LIN {X 0,Y 575.439,Z 360.454,A -85,B 0,C 180,E1 -10255.385,E2 -10255.385} C_VEL
LIN {X 0,Y 575.391,Z 376.581,A -85,B 0,C 180,E1 -10255.636,E2 -10255.636} C_VEL
LIN {X 0,Y 573.804,Z 481.536,A -85,B 0,C 180,E1 -10257.179,E2 -10257.179} C_VEL
LIN {X 0,Y 573.47,Z 496.036,A -85,B 0,C 180,E1 -10257.528,E2 -10257.528} C_VEL
LIN {X 0,Y 572.934,Z 510.451,A -85,B 0,C 180,E1 -10258.03,E2 -10258.03} C_VEL
LIN {X 0,Y 572.466,Z 522.841,A -85,B 0,C 180,E1 -10258.598,E2 -10258.598} C_VEL
LIN {X 0,Y 571.889,Z 535.06,A -85,B 0,C 180,E1 -10259.298,E2 -10259.298} C_VEL
LIN {X 0,Y 571.402,Z 547.39,A -85,B 0,C 180,E1 -10260.176,E2 -10260.176} C_VEL
LIN {X 0,Y 570.935,Z 557.583,A -85,B 0,C 180,E1 -10261.054,E2 -10261.054} C_VEL
LIN {X 0,Y 570.32,Z 567.822,A -85,B 0,C 180,E1 -10262.112,E2 -10262.112} C_VEL
LIN {X 0,Y 569.977,Z 576.267,A -85,B 0,C 180,E1 -10263.17,E2 -10263.17} C_VEL
LIN {X 0,Y 569.621,Z 583.313,A -85,B 0,C 180,E1 -10264.231,E2 -10264.231} C_VEL
LIN {X 0,Y 569.503,Z 588.963,A -85,B 0,C 180,E1 -10265.257,E2 -10265.257} C_VEL
LIN {X 0,Y 569.323,Z 593.962,A -85,B 0,C 180,E1 -10266.357,E2 -10266.357} C_VEL
LIN {X 0,Y 569.1,Z 598.933,A -85,B 0,C 180,E1 -10267.781,E2 -10267.781} C_VEL
LIN {X 0,Y 569.035,Z 602.372,A -85,B 0,C 180,E1 -10269.208,E2 -10269.208} C_VEL
LIN {X 0,Y 569.056,Z 603.678,A -85,B 0,C 180,E1 -10270.028,E2 -10270.028} C_VEL
LIN {X 0,Y 568.925,Z 604.796,A -85,B 0,C 180,E1 -10271.361,E2 -10271.361} C_VEL
LIN {X 0,Y 568.971,Z 604.604,A -85,B 0,C 180,E1 -10272.803,E2 -10272.803} C_VEL
LIN {X 0,Y 569.033,Z 603.97,A -85,B 0,C 180,E1 -10273.526,E2 -10273.526} C_VEL
LIN {X 0,Y 568.978,Z 601.595,A -85,B 0,C 180,E1 -10274.982,E2 -10274.982} C_VEL
LIN {X 0,Y 569.112,Z 597.684,A -85,B 0,C 180,E1 -10276.444,E2 -10276.444} C_VEL
LIN {X 0,Y 569.206,Z 593.593,A -85,B 0,C 180,E1 -10277.547,E2 -10277.547} C_VEL
LIN {X 0,Y 569.387,Z 588.256,A -85,B 0,C 180,E1 -10278.693,E2 -10278.693} C_VEL
LIN {X 0,Y 569.633,Z 580.967,A -85,B 0,C 180,E1 -10279.952,E2 -10279.952} C_VEL
LIN {X 0,Y 569.942,Z 573.158,A -85,B 0,C 180,E1 -10281.049,E2 -10281.049} C_VEL
LIN {X 0,Y 570.356,Z 563.337,A -85,B 0,C 180,E1 -10282.187,E2 -10282.187} C_VEL
LIN {X 0,Y 570.787,Z 552.451,A -85,B 0,C 180,E1 -10283.218,E2 -10283.218} C_VEL
LIN {X 0,Y 571.326,Z 540.367,A -85,B 0,C 180,E1 -10284.153,E2 -10284.153} C_VEL
LIN {X 0,Y 571.808,Z 527.265,A -85,B 0,C 180,E1 -10284.976,E2 -10284.976} C_VEL
LIN {X 0,Y 572.223,Z 514.526,A -85,B 0,C 180,E1 -10285.611,E2 -10285.611} C_VEL
LIN {X 0,Y 572.651,Z 501.122,A -85,B 0,C 180,E1 -10286.125,E2 -10286.125} C_VEL
LIN {X 0,Y 573.109,Z 487.002,A -85,B 0,C 180,E1 -10286.518,E2 -10286.518} C_VEL
LIN {X 0,Y 573.287,Z 471.7,A -85,B 0,C 180,E1 -10286.795,E2 -10286.795} C_VEL
LIN {X 0,Y 574.437,Z 360.487,A -85,B 0,C 180,E1 -10288.346,E2 -10288.346} C_VEL
LIN {X 0,Y 571.59,Z 342.196,A -85,B 0,C 180,E1 -10288.699,E2 -10288.699} C_VEL
LIN {X 0,Y 572.257,Z 318.728,A -85,B 0,C 180,E1 -10291.757,E2 -10291.757} C_VEL
LIN {X 0,Y 572.767,Z 299.778,A -85,B 0,C 180,E1 -10294.232,E2 -10294.232} C_VEL
LIN {X 0,Y 571.08,Z 289.612,A -85,B 0,C 180,E1 -10295.634,E2 -10295.634} C_VEL
LIN {X 0,Y 570.357,Z 286,A -85,B 0,C 180,E1 -10296.147,E2 -10296.147} C_VEL
LIN {X 0,Y 570.263,Z 286.005,A -85,B 0,C 180,E1 -10299.3,E2 -10299.3} C_VEL
LIN {X 0,Y 570.28,Z 286.004,A -85,B 0,C 180,E1 -10301.548,E2 -10301.548} C_VEL
LIN {X 0,Y 570.317,Z 286.001,A -85,B 0,C 180,E1 -10304.573,E2 -10304.573} C_VEL
LIN {X 0,Y 570.263,Z 286.007,A -85,B 0,C 180,E1 -10307.501,E2 -10307.501} C_VEL
LIN {X 0,Y 570.283,Z 286.006,A -85,B 0,C 180,E1 -10310.305,E2 -10310.305} C_VEL
LIN {X 0,Y 570.273,Z 286.007,A -85,B 0,C 180,E1 -10312.996,E2 -10312.996} C_VEL
LIN {X 0,Y 570.287,Z 286.006,A -85,B 0,C 180,E1 -10315.597,E2 -10315.597} C_VEL
LIN {X 0,Y 570.315,Z 286.001,A -85,B 0,C 180,E1 -10318.121,E2 -10318.121} C_VEL
LIN {X 0,Y 570.294,Z 286.005,A -85,B 0,C 180,E1 -10321.378,E2 -10321.378} C_VEL
LIN {X 0,Y 570.293,Z 286.004,A -85,B 0,C 180,E1 -10322.089,E2 -10322.089} C_VEL
LIN {X 0,Y 569.657,Z 286.086,A -85,B 0,C 180,E1 -10322.678,E2 -10322.678} C_VEL
LIN {X 0,Y 566.811,Z 286.439,A -85,B 0,C 180,E1 -10323.635,E2 -10323.635} C_VEL
LIN {X 0,Y 564.388,Z 286.742,A -85,B 0,C 180,E1 -10324.404,E2 -10324.404} C_VEL
LIN {X 0,Y 563.349,Z 286.869,A -85,B 0,C 180,E1 -10324.999,E2 -10324.999} C_VEL
LIN {X 0,Y 563.267,Z 286.879,A -85,B 0,C 180,E1 -10325.2,E2 -10325.2} C_VEL
LIN {X 0,Y 563.302,Z 286.876,A -85,B 0,C 180,E1 -10328.095,E2 -10328.095} C_VEL
LIN {X 0,Y 563.305,Z 286.874,A -85,B 0,C 180,E1 -10331.136,E2 -10331.136} C_VEL
LIN {X 0,Y 563.311,Z 286.878,A -85,B 0,C 180,E1 -10334.122,E2 -10334.122} C_VEL
LIN {X 0,Y 563.359,Z 286.869,A -85,B 0,C 180,E1 -10336.334,E2 -10336.334} C_VEL
LIN {X 0,Y 563.372,Z 286.864,A -85,B 0,C 180,E1 -10339.25,E2 -10339.25} C_VEL
LIN {X 0,Y 563.397,Z 286.866,A -85,B 0,C 180,E1 -10342.497,E2 -10342.497} C_VEL
LIN {X 0,Y 563.431,Z 286.922,A -85,B 0,C 180,E1 -10342.857,E2 -10342.857} C_VEL
LIN {X 0,Y 564.572,Z 294.675,A -85,B 0,C 180,E1 -10344.302,E2 -10344.302} C_VEL
LIN {X 0,Y 564.436,Z 300.116,A -85,B 0,C 180,E1 -10345.271,E2 -10345.271} C_VEL
LIN {X 0,Y 567.828,Z 316.778,A -85,B 0,C 180,E1 -10345.577,E2 -10345.577} C_VEL
LIN {X 0,Y 566.808,Z 435.74,A -85,B 0,C 180,E1 -10347.099,E2 -10347.099} C_VEL
LIN {X 0,Y 566.508,Z 450.139,A -85,B 0,C 180,E1 -10347.429,E2 -10347.429} C_VEL
LIN {X 0,Y 566.207,Z 463.339,A -85,B 0,C 180,E1 -10347.871,E2 -10347.871} C_VEL
LIN {X 0,Y 565.821,Z 475.423,A -85,B 0,C 180,E1 -10348.402,E2 -10348.402} C_VEL
LIN {X 0,Y 565.416,Z 488.106,A -85,B 0,C 180,E1 -10349.111,E2 -10349.111} C_VEL
LIN {X 0,Y 564.727,Z 499.728,A -85,B 0,C 180,E1 -10349.909,E2 -10349.909} C_VEL
LIN {X 0,Y 564.286,Z 511.265,A -85,B 0,C 180,E1 -10350.887,E2 -10350.887} C_VEL
LIN {X 0,Y 563.681,Z 521.642,A -85,B 0,C 180,E1 -10351.957,E2 -10351.957} C_VEL
LIN {X 0,Y 563.288,Z 530.194,A -85,B 0,C 180,E1 -10353.028,E2 -10353.028} C_VEL
LIN {X 0,Y 562.818,Z 538.433,A -85,B 0,C 180,E1 -10354.281,E2 -10354.281} C_VEL
LIN {X 0,Y 562.684,Z 544.812,A -85,B 0,C 180,E1 -10355.488,E2 -10355.488} C_VEL
LIN {X 0,Y 562.439,Z 550.296,A -85,B 0,C 180,E1 -10356.793,E2 -10356.793} C_VEL
LIN {X 0,Y 562.242,Z 553.805,A -85,B 0,C 180,E1 -10357.875,E2 -10357.875} C_VEL
LIN {X 0,Y 562.144,Z 557.231,A -85,B 0,C 180,E1 -10359.32,E2 -10359.32} C_VEL
LIN {X 0,Y 562.095,Z 559.271,A -85,B 0,C 180,E1 -10360.771,E2 -10360.771} C_VEL
LIN {X 0,Y 562.043,Z 559.951,A -85,B 0,C 180,E1 -10362.229,E2 -10362.229} C_VEL
LIN {X 0,Y 562.154,Z 559.253,A -85,B 0,C 180,E1 -10363.692,E2 -10363.692} C_VEL
LIN {X 0,Y 562.211,Z 557.174,A -85,B 0,C 180,E1 -10365.165,E2 -10365.165} C_VEL
LIN {X 0,Y 562.424,Z 553.635,A -85,B 0,C 180,E1 -10366.643,E2 -10366.643} C_VEL
LIN {X 0,Y 562.685,Z 548.511,A -85,B 0,C 180,E1 -10368.13,E2 -10368.13} C_VEL
LIN {X 0,Y 563.038,Z 542.646,A -85,B 0,C 180,E1 -10369.418,E2 -10369.418} C_VEL
LIN {X 0,Y 563.498,Z 535.031,A -85,B 0,C 180,E1 -10370.746,E2 -10370.746} C_VEL
LIN {X 0,Y 564.017,Z 527.054,A -85,B 0,C 180,E1 -10371.872,E2 -10371.872} C_VEL
LIN {X 0,Y 564.601,Z 517.329,A -85,B 0,C 180,E1 -10373.001,E2 -10373.001} C_VEL
LIN {X 0,Y 565.263,Z 506.553,A -85,B 0,C 180,E1 -10374.028,E2 -10374.028} C_VEL
LIN {X 0,Y 565.934,Z 494.604,A -85,B 0,C 180,E1 -10374.958,E2 -10374.958} C_VEL
LIN {X 0,Y 566.519,Z 482.243,A -85,B 0,C 180,E1 -10375.737,E2 -10375.737} C_VEL
LIN {X 0,Y 567.105,Z 468.979,A -85,B 0,C 180,E1 -10376.398,E2 -10376.398} C_VEL
LIN {X 0,Y 567.526,Z 456.619,A -85,B 0,C 180,E1 -10376.871,E2 -10376.871} C_VEL
LIN {X 0,Y 567.835,Z 442.693,A -85,B 0,C 180,E1 -10377.263,E2 -10377.263} C_VEL
LIN {X 0,Y 567.93,Z 427.921,A -85,B 0,C 180,E1 -10377.524,E2 -10377.524} C_VEL
LIN {X 0,Y 569.043,Z 317.141,A -85,B 0,C 180,E1 -10378.943,E2 -10378.943} C_VEL
LIN {X 0,Y 565.232,Z 300.482,A -85,B 0,C 180,E1 -10379.325,E2 -10379.325} C_VEL
LIN {X 0,Y 565.026,Z 296.096,A -85,B 0,C 180,E1 -10380.146,E2 -10380.146} C_VEL
LIN {X 0,Y 563.228,Z 286.887,A -85,B 0,C 180,E1 -10381.992,E2 -10381.992} C_VEL
LIN {X 0,Y 563.243,Z 286.882,A -85,B 0,C 180,E1 -10384.891,E2 -10384.891} C_VEL
LIN {X 0,Y 563.207,Z 286.886,A -85,B 0,C 180,E1 -10387.543,E2 -10387.543} C_VEL
LIN {X 0,Y 563.226,Z 286.882,A -85,B 0,C 180,E1 -10390.658,E2 -10390.658} C_VEL
LIN {X 0,Y 563.238,Z 286.882,A -85,B 0,C 180,E1 -10393.152,E2 -10393.152} C_VEL
LIN {X 0,Y 563.232,Z 286.879,A -85,B 0,C 180,E1 -10395.859,E2 -10395.859} C_VEL
LIN {X 0,Y 563.227,Z 286.882,A -85,B 0,C 180,E1 -10398.767,E2 -10398.767} C_VEL
LIN {X 0,Y 563.249,Z 286.883,A -85,B 0,C 180,E1 -10401.574,E2 -10401.574} C_VEL
LIN {X 0,Y 563.273,Z 286.863,A -85,B 0,C 180,E1 -10404.235,E2 -10404.235} C_VEL
LIN {X 0,Y 563.205,Z 286.883,A -85,B 0,C 180,E1 -10406.824,E2 -10406.824} C_VEL
LIN {X 0,Y 563.26,Z 286.877,A -85,B 0,C 180,E1 -10409.346,E2 -10409.346} C_VEL
LIN {X 0,Y 563.269,Z 286.875,A -85,B 0,C 180,E1 -10411.99,E2 -10411.99} C_VEL
LIN {X 0,Y 563.24,Z 286.883,A -85,B 0,C 180,E1 -10415.201,E2 -10415.201} C_VEL
LIN {X 0,Y 563.275,Z 286.876,A -85,B 0,C 180,E1 -10418.096,E2 -10418.096} C_VEL
LIN {X 0,Y 563.274,Z 286.874,A -85,B 0,C 180,E1 -10421.136,E2 -10421.136} C_VEL
LIN {X 0,Y 563.269,Z 286.875,A -85,B 0,C 180,E1 -10424.123,E2 -10424.123} C_VEL
LIN {X 0,Y 563.341,Z 286.86,A -85,B 0,C 180,E1 -10426.335,E2 -10426.335} C_VEL
LIN {X 0,Y 563.343,Z 286.873,A -85,B 0,C 180,E1 -10429.251,E2 -10429.251} C_VEL
LIN {X 0,Y 563.367,Z 286.86,A -85,B 0,C 180,E1 -10432.139,E2 -10432.139} C_VEL
LIN {X 0,Y 563.439,Z 286.86,A -85,B 0,C 180,E1 -10435.008,E2 -10435.008} C_VEL
LIN {X 0,Y 563.447,Z 286.854,A -85,B 0,C 180,E1 -10438.575,E2 -10438.575} C_VEL
LIN {X 0,Y 563.573,Z 286.836,A -85,B 0,C 180,E1 -10440,E2 -10440} C_VEL
LIN {X 0,Y 563.303,Z 286.862,A -85,B 0,C 180,E1 -10442.138,E2 -10442.138} C_VEL
LIN {X 0,Y 563.455,Z 286.86,A -85,B 0,C 180,E1 -10444.992,E2 -10444.992} C_VEL
LIN {X 0,Y 563.368,Z 286.855,A -85,B 0,C 180,E1 -10447.861,E2 -10447.861} C_VEL
LIN {X 0,Y 563.392,Z 286.864,A -85,B 0,C 180,E1 -10450.848,E2 -10450.848} C_VEL
LIN {X 0,Y 563.349,Z 286.862,A -85,B 0,C 180,E1 -10454.123,E2 -10454.123} C_VEL
LIN {X 0,Y 563.319,Z 286.868,A -85,B 0,C 180,E1 -10456.786,E2 -10456.786} C_VEL
LIN {X 0,Y 563.26,Z 286.875,A -85,B 0,C 180,E1 -10459.619,E2 -10459.619} C_VEL
LIN {X 0,Y 563.275,Z 286.869,A -85,B 0,C 180,E1 -10461.904,E2 -10461.904} C_VEL
LIN {X 0,Y 563.24,Z 286.883,A -85,B 0,C 180,E1 -10464.8,E2 -10464.8} C_VEL
LIN {X 0,Y 563.269,Z 286.876,A -85,B 0,C 180,E1 -10468.01,E2 -10468.01} C_VEL
LIN {X 0,Y 563.261,Z 286.879,A -85,B 0,C 180,E1 -10470.907,E2 -10470.907} C_VEL
LIN {X 0,Y 563.237,Z 286.877,A -85,B 0,C 180,E1 -10473.574,E2 -10473.574} C_VEL
LIN {X 0,Y 563.309,Z 286.856,A -85,B 0,C 180,E1 -10476.08,E2 -10476.08} C_VEL
LIN {X 0,Y 563.3,Z 286.879,A -85,B 0,C 180,E1 -10478.443,E2 -10478.443} C_VEL
LIN {X 0,Y 563.243,Z 286.879,A -85,B 0,C 180,E1 -10481.232,E2 -10481.232} C_VEL
LIN {X 0,Y 563.228,Z 286.883,A -85,B 0,C 180,E1 -10483.841,E2 -10483.841} C_VEL
LIN {X 0,Y 563.233,Z 286.887,A -85,B 0,C 180,E1 -10486.162,E2 -10486.162} C_VEL
LIN {X 0,Y 563.264,Z 286.877,A -85,B 0,C 180,E1 -10488.773,E2 -10488.773} C_VEL
LIN {X 0,Y 563.285,Z 286.876,A -85,B 0,C 180,E1 -10491.573,E2 -10491.573} C_VEL
LIN {X 0,Y 563.303,Z 286.877,A -85,B 0,C 180,E1 -10494.24,E2 -10494.24} C_VEL
LIN {X 0,Y 563.244,Z 286.884,A -85,B 0,C 180,E1 -10496.829,E2 -10496.829} C_VEL
LIN {X 0,Y 563.266,Z 286.884,A -85,B 0,C 180,E1 -10499.349,E2 -10499.349} C_VEL
LIN {X 0,Y 563.289,Z 286.879,A -85,B 0,C 180,E1 -10502.516,E2 -10502.516} C_VEL
LIN {X 0,Y 566.847,Z 303.208,A -85,B 0,C 180,E1 -10505.009,E2 -10505.009} C_VEL
LIN {X 0,Y 567.241,Z 307.117,A -85,B 0,C 180,E1 -10505.567,E2 -10505.567} C_VEL
LIN {X 0,Y 566.095,Z 326.832,A -85,B 0,C 180,E1 -10508.213,E2 -10508.213} C_VEL
LIN {X 0,Y 564.836,Z 350.849,A -85,B 0,C 180,E1 -10511.38,E2 -10511.38} C_VEL
LIN {X 0,Y 564.394,Z 361.151,A -85,B 0,C 180,E1 -10512.71,E2 -10512.71} C_VEL
LIN {X 0,Y 567.671,Z 382.814,A -85,B 0,C 180,E1 -10513.112,E2 -10513.112} C_VEL
LIN {X 0,Y 568.575,Z 391.391,A -85,B 0,C 180,E1 -10513.255,E2 -10513.255} C_VEL
LIN {X 0,Y 567.497,Z 499.318,A -85,B 0,C 180,E1 -10514.651,E2 -10514.651} C_VEL
LIN {X 0,Y 566.972,Z 514.115,A -85,B 0,C 180,E1 -10514.988,E2 -10514.988} C_VEL
LIN {X 0,Y 566.391,Z 527.966,A -85,B 0,C 180,E1 -10515.453,E2 -10515.453} C_VEL
LIN {X 0,Y 565.747,Z 540.9,A -85,B 0,C 180,E1 -10516.031,E2 -10516.031} C_VEL
LIN {X 0,Y 565.032,Z 553.471,A -85,B 0,C 180,E1 -10516.744,E2 -10516.744} C_VEL
LIN {X 0,Y 564.367,Z 564.958,A -85,B 0,C 180,E1 -10517.549,E2 -10517.549} C_VEL
LIN {X 0,Y 563.709,Z 576.506,A -85,B 0,C 180,E1 -10518.535,E2 -10518.535} C_VEL
LIN {X 0,Y 563.228,Z 586.869,A -85,B 0,C 180,E1 -10519.613,E2 -10519.613} C_VEL
LIN {X 0,Y 562.765,Z 595.446,A -85,B 0,C 180,E1 -10520.69,E2 -10520.69} C_VEL
LIN {X 0,Y 562.348,Z 603.685,A -85,B 0,C 180,E1 -10521.947,E2 -10521.947} C_VEL
LIN {X 0,Y 562.143,Z 612.58,A -85,B 0,C 180,E1 -10523.563,E2 -10523.563} C_VEL
LIN {X 0,Y 562.068,Z 617.376,A -85,B 0,C 180,E1 -10524.639,E2 -10524.639} C_VEL
LIN {X 0,Y 561.972,Z 621.998,A -85,B 0,C 180,E1 -10525.971,E2 -10525.971} C_VEL
LIN {X 0,Y 562.009,Z 624.928,A -85,B 0,C 180,E1 -10527.144,E2 -10527.144} C_VEL
LIN {X 0,Y 561.962,Z 627.166,A -85,B 0,C 180,E1 -10528.573,E2 -10528.573} C_VEL
LIN {X 0,Y 561.985,Z 627.985,A -85,B 0,C 180,E1 -10530.002,E2 -10530.002} C_VEL
LIN {X 0,Y 561.961,Z 627.392,A -85,B 0,C 180,E1 -10531.43,E2 -10531.43} C_VEL
LIN {X 0,Y 562.011,Z 625.363,A -85,B 0,C 180,E1 -10532.859,E2 -10532.859} C_VEL
LIN {X 0,Y 562.019,Z 621.854,A -85,B 0,C 180,E1 -10534.29,E2 -10534.29} C_VEL
LIN {X 0,Y 562.073,Z 618.238,A -85,B 0,C 180,E1 -10535.365,E2 -10535.365} C_VEL
LIN {X 0,Y 562.151,Z 613.624,A -85,B 0,C 180,E1 -10536.44,E2 -10536.44} C_VEL
LIN {X 0,Y 562.339,Z 606.953,A -85,B 0,C 180,E1 -10537.697,E2 -10537.697} C_VEL
LIN {X 0,Y 562.664,Z 598.641,A -85,B 0,C 180,E1 -10538.954,E2 -10538.954} C_VEL
LIN {X 0,Y 562.963,Z 589.911,A -85,B 0,C 180,E1 -10540.033,E2 -10540.033} C_VEL
LIN {X 0,Y 563.464,Z 580.417,A -85,B 0,C 180,E1 -10541.011,E2 -10541.011} C_VEL
LIN {X 0,Y 563.945,Z 568.675,A -85,B 0,C 180,E1 -10542.009,E2 -10542.009} C_VEL
LIN {X 0,Y 564.465,Z 557.07,A -85,B 0,C 180,E1 -10542.817,E2 -10542.817} C_VEL
LIN {X 0,Y 565.06,Z 544.353,A -85,B 0,C 180,E1 -10543.533,E2 -10543.533} C_VEL
LIN {X 0,Y 565.545,Z 531.258,A -85,B 0,C 180,E1 -10544.115,E2 -10544.115} C_VEL
LIN {X 0,Y 566.049,Z 517.241,A -85,B 0,C 180,E1 -10544.582,E2 -10544.582} C_VEL
LIN {X 0,Y 566.5,Z 499.468,A -85,B 0,C 180,E1 -10544.982,E2 -10544.982} C_VEL
LIN {X 0,Y 567.554,Z 424.5,A -85,B 0,C 180,E1 -10546.077,E2 -10546.077} C_VEL
LIN {X 0,Y 568.068,Z 389.136,A -85,B 0,C 180,E1 -10546.623,E2 -10546.623} C_VEL
LIN {X 0,Y 564.86,Z 363.019,A -85,B 0,C 180,E1 -10547.174,E2 -10547.174} C_VEL
LIN {X 0,Y 564.089,Z 357.909,A -85,B 0,C 180,E1 -10547.295,E2 -10547.295} C_VEL
LIN {X 0,Y 564.97,Z 335.865,A -85,B 0,C 180,E1 -10550.125,E2 -10550.125} C_VEL
LIN {X 0,Y 566.057,Z 312.595,A -85,B 0,C 180,E1 -10553.135,E2 -10553.135} C_VEL
LIN {X 0,Y 566.375,Z 302.386,A -85,B 0,C 180,E1 -10554.477,E2 -10554.477} C_VEL
LIN {X 0,Y 563.285,Z 286.88,A -85,B 0,C 180,E1 -10556.695,E2 -10556.695} C_VEL
LIN {X 0,Y 563.254,Z 286.883,A -85,B 0,C 180,E1 -10559.483,E2 -10559.483} C_VEL
LIN {X 0,Y 563.247,Z 286.878,A -85,B 0,C 180,E1 -10562.328,E2 -10562.328} C_VEL
LIN {X 0,Y 563.261,Z 286.879,A -85,B 0,C 180,E1 -10564.894,E2 -10564.894} C_VEL
LIN {X 0,Y 563.204,Z 286.892,A -85,B 0,C 180,E1 -10567.548,E2 -10567.548} C_VEL
LIN {X 0,Y 563.245,Z 286.88,A -85,B 0,C 180,E1 -10570.66,E2 -10570.66} C_VEL
LIN {X 0,Y 563.226,Z 286.883,A -85,B 0,C 180,E1 -10573.838,E2 -10573.838} C_VEL
LIN {X 0,Y 563.24,Z 286.88,A -85,B 0,C 180,E1 -10576.162,E2 -10576.162} C_VEL
LIN {X 0,Y 563.246,Z 286.882,A -85,B 0,C 180,E1 -10579.341,E2 -10579.341} C_VEL
LIN {X 0,Y 563.227,Z 286.886,A -85,B 0,C 180,E1 -10582.455,E2 -10582.455} C_VEL
LIN {X 0,Y 563.276,Z 286.879,A -85,B 0,C 180,E1 -10585.159,E2 -10585.159} C_VEL
LIN {X 0,Y 563.252,Z 286.879,A -85,B 0,C 180,E1 -10587.741,E2 -10587.741} C_VEL
LIN {X 0,Y 563.257,Z 286.884,A -85,B 0,C 180,E1 -10590.518,E2 -10590.518} C_VEL
LIN {X 0,Y 563.276,Z 286.881,A -85,B 0,C 180,E1 -10592.606,E2 -10592.606} C_VEL
LIN {X 0,Y 563.268,Z 286.882,A -85,B 0,C 180,E1 -10595.772,E2 -10595.772} C_VEL
LIN {X 0,Y 563.305,Z 286.883,A -85,B 0,C 180,E1 -10598.097,E2 -10598.097} C_VEL
LIN {X 0,Y 563.305,Z 286.879,A -85,B 0,C 180,E1 -10601.137,E2 -10601.137} C_VEL
LIN {X 0,Y 563.291,Z 286.879,A -85,B 0,C 180,E1 -10604.123,E2 -10604.123} C_VEL
LIN {X 0,Y 563.362,Z 286.871,A -85,B 0,C 180,E1 -10606.336,E2 -10606.336} C_VEL
LIN {X 0,Y 563.322,Z 286.946,A -85,B 0,C 180,E1 -10607.272,E2 -10607.272} C_VEL
LIN {X 0,Y 566.211,Z 300.084,A -85,B 0,C 180,E1 -10609.126,E2 -10609.126} C_VEL
LIN {X 0,Y 566.493,Z 305.5,A -85,B 0,C 180,E1 -10609.852,E2 -10609.852} C_VEL
LIN {X 0,Y 566.027,Z 325.116,A -85,B 0,C 180,E1 -10612.38,E2 -10612.38} C_VEL
LIN {X 0,Y 565.383,Z 343.211,A -85,B 0,C 180,E1 -10614.713,E2 -10614.713} C_VEL
LIN {X 0,Y 568.329,Z 358.791,A -85,B 0,C 180,E1 -10615.095,E2 -10615.095} C_VEL
LIN {X 0,Y 568.96,Z 363.16,A -85,B 0,C 180,E1 -10615.189,E2 -10615.189} C_VEL
LIN {X 0,Y 566.993,Z 482.592,A -85,B 0,C 180,E1 -10616.99,E2 -10616.99} C_VEL
LIN {X 0,Y 566.647,Z 496.712,A -85,B 0,C 180,E1 -10617.343,E2 -10617.343} C_VEL
LIN {X 0,Y 566.103,Z 510.414,A -85,B 0,C 180,E1 -10617.828,E2 -10617.828} C_VEL
LIN {X 0,Y 565.619,Z 522.816,A -85,B 0,C 180,E1 -10618.403,E2 -10618.403} C_VEL
LIN {X 0,Y 565.016,Z 535.052,A -85,B 0,C 180,E1 -10619.112,E2 -10619.112} C_VEL
LIN {X 0,Y 564.472,Z 547.43,A -85,B 0,C 180,E1 -10620,E2 -10620} C_VEL
LIN {X 0,Y 563.987,Z 557.648,A -85,B 0,C 180,E1 -10620.889,E2 -10620.889} C_VEL
LIN {X 0,Y 563.341,Z 567.899,A -85,B 0,C 180,E1 -10621.959,E2 -10621.959} C_VEL
LIN {X 0,Y 562.98,Z 576.351,A -85,B 0,C 180,E1 -10623.031,E2 -10623.031} C_VEL
LIN {X 0,Y 562.559,Z 583.414,A -85,B 0,C 180,E1 -10624.105,E2 -10624.105} C_VEL
LIN {X 0,Y 562.426,Z 590.153,A -85,B 0,C 180,E1 -10625.359,E2 -10625.359} C_VEL
LIN {X 0,Y 562.248,Z 594.798,A -85,B 0,C 180,E1 -10626.438,E2 -10626.438} C_VEL
LIN {X 0,Y 562,Z 599.608,A -85,B 0,C 180,E1 -10627.88,E2 -10627.88} C_VEL
LIN {X 0,Y 561.951,Z 602.845,A -85,B 0,C 180,E1 -10629.325,E2 -10629.325} C_VEL
LIN {X 0,Y 561.981,Z 603.908,A -85,B 0,C 180,E1 -10630.049,E2 -10630.049} C_VEL
LIN {X 0,Y 561.835,Z 604.982,A -85,B 0,C 180,E1 -10631.506,E2 -10631.506} C_VEL
LIN {X 0,Y 561.895,Z 604.625,A -85,B 0,C 180,E1 -10632.967,E2 -10632.967} C_VEL
LIN {X 0,Y 561.926,Z 603.906,A -85,B 0,C 180,E1 -10633.7,E2 -10633.7} C_VEL
LIN {X 0,Y 561.893,Z 601.356,A -85,B 0,C 180,E1 -10635.176,E2 -10635.176} C_VEL
LIN {X 0,Y 562.031,Z 598.235,A -85,B 0,C 180,E1 -10636.333,E2 -10636.333} C_VEL
LIN {X 0,Y 562.172,Z 592.965,A -85,B 0,C 180,E1 -10637.774,E2 -10637.774} C_VEL
LIN {X 0,Y 562.418,Z 586.621,A -85,B 0,C 180,E1 -10639.082,E2 -10639.082} C_VEL
LIN {X 0,Y 562.606,Z 579.844,A -85,B 0,C 180,E1 -10640.212,E2 -10640.212} C_VEL
LIN {X 0,Y 562.972,Z 571.595,A -85,B 0,C 180,E1 -10641.341,E2 -10641.341} C_VEL
LIN {X 0,Y 563.415,Z 561.525,A -85,B 0,C 180,E1 -10642.475,E2 -10642.475} C_VEL
LIN {X 0,Y 563.868,Z 550.24,A -85,B 0,C 180,E1 -10643.519,E2 -10643.519} C_VEL
LIN {X 0,Y 564.359,Z 538.998,A -85,B 0,C 180,E1 -10644.373,E2 -10644.373} C_VEL
LIN {X 0,Y 564.845,Z 526.629,A -85,B 0,C 180,E1 -10645.141,E2 -10645.141} C_VEL
LIN {X 0,Y 565.291,Z 513.254,A -85,B 0,C 180,E1 -10645.8,E2 -10645.8} C_VEL
LIN {X 0,Y 565.727,Z 499.409,A -85,B 0,C 180,E1 -10646.321,E2 -10646.321} C_VEL
LIN {X 0,Y 566.171,Z 484.533,A -85,B 0,C 180,E1 -10646.72,E2 -10646.72} C_VEL
LIN {X 0,Y 566.376,Z 467.777,A -85,B 0,C 180,E1 -10646.998,E2 -10646.998} C_VEL
LIN {X 0,Y 567.563,Z 361.331,A -85,B 0,C 180,E1 -10648.508,E2 -10648.508} C_VEL
LIN {X 0,Y 564.62,Z 342.226,A -85,B 0,C 180,E1 -10648.887,E2 -10648.887} C_VEL
LIN {X 0,Y 565.275,Z 320.222,A -85,B 0,C 180,E1 -10651.778,E2 -10651.778} C_VEL
LIN {X 0,Y 565.83,Z 301.104,A -85,B 0,C 180,E1 -10654.289,E2 -10654.289} C_VEL
LIN {X 0,Y 563.894,Z 289.819,A -85,B 0,C 180,E1 -10655.85,E2 -10655.85} C_VEL
LIN {X 0,Y 563.304,Z 286.879,A -85,B 0,C 180,E1 -10656.295,E2 -10656.295} C_VEL
LIN {X 0,Y 563.234,Z 286.882,A -85,B 0,C 180,E1 -10659.551,E2 -10659.551} C_VEL
LIN {X 0,Y 563.269,Z 286.883,A -85,B 0,C 180,E1 -10662.184,E2 -10662.184} C_VEL
LIN {X 0,Y 563.278,Z 286.877,A -85,B 0,C 180,E1 -10665.138,E2 -10665.138} C_VEL
LIN {X 0,Y 563.212,Z 286.887,A -85,B 0,C 180,E1 -10668.262,E2 -10668.262} C_VEL
LIN {X 0,Y 563.219,Z 286.885,A -85,B 0,C 180,E1 -10670.634,E2 -10670.634} C_VEL
LIN {X 0,Y 563.257,Z 286.883,A -85,B 0,C 180,E1 -10673.932,E2 -10673.932} C_VEL
LIN {X 0,Y 563.228,Z 286.885,A -85,B 0,C 180,E1 -10676.824,E2 -10676.824} C_VEL
LIN {X 0,Y 563.25,Z 286.882,A -85,B 0,C 180,E1 -10679.344,E2 -10679.344} C_VEL
LIN {X 0,Y 563.264,Z 286.879,A -85,B 0,C 180,E1 -10682.085,E2 -10682.085} C_VEL
LIN {X 0,Y 563.267,Z 286.879,A -85,B 0,C 180,E1 -10685.2,E2 -10685.2} C_VEL
LIN {X 0,Y 562.602,Z 286.963,A -85,B 0,C 180,E1 -10685.797,E2 -10685.797} C_VEL
LIN {X 0,Y 559.742,Z 287.318,A -85,B 0,C 180,E1 -10686.765,E2 -10686.765} C_VEL
LIN {X 0,Y 557.333,Z 287.618,A -85,B 0,C 180,E1 -10687.545,E2 -10687.545} C_VEL
LIN {X 0,Y 556.313,Z 287.747,A -85,B 0,C 180,E1 -10688.147,E2 -10688.147} C_VEL
LIN {X 0,Y 556.237,Z 287.754,A -85,B 0,C 180,E1 -10688.351,E2 -10688.351} C_VEL
LIN {X 0,Y 556.252,Z 287.752,A -85,B 0,C 180,E1 -10690.888,E2 -10690.888} C_VEL
LIN {X 0,Y 556.264,Z 287.753,A -85,B 0,C 180,E1 -10693.916,E2 -10693.916} C_VEL
LIN {X 0,Y 556.328,Z 287.747,A -85,B 0,C 180,E1 -10696.158,E2 -10696.158} C_VEL
LIN {X 0,Y 556.361,Z 287.737,A -85,B 0,C 180,E1 -10699.113,E2 -10699.113} C_VEL
LIN {X 0,Y 556.362,Z 287.742,A -85,B 0,C 180,E1 -10702.584,E2 -10702.584} C_VEL
LIN {X 0,Y 556.394,Z 287.963,A -85,B 0,C 180,E1 -10702.766,E2 -10702.766} C_VEL
LIN {X 0,Y 557.579,Z 295.744,A -85,B 0,C 180,E1 -10704.23,E2 -10704.23} C_VEL
LIN {X 0,Y 557.47,Z 300.601,A -85,B 0,C 180,E1 -10705.088,E2 -10705.088} C_VEL
LIN {X 0,Y 561.01,Z 318.615,A -85,B 0,C 180,E1 -10705.42,E2 -10705.42} C_VEL
LIN {X 0,Y 559.91,Z 435.507,A -85,B 0,C 180,E1 -10706.928,E2 -10706.928} C_VEL
LIN {X 0,Y 559.596,Z 450.147,A -85,B 0,C 180,E1 -10707.263,E2 -10707.263} C_VEL
LIN {X 0,Y 559.284,Z 463.452,A -85,B 0,C 180,E1 -10707.71,E2 -10707.71} C_VEL
LIN {X 0,Y 558.859,Z 476.471,A -85,B 0,C 180,E1 -10708.293,E2 -10708.293} C_VEL
LIN {X 0,Y 558.412,Z 489.045,A -85,B 0,C 180,E1 -10709.01,E2 -10709.01} C_VEL
LIN {X 0,Y 557.725,Z 500.573,A -85,B 0,C 180,E1 -10709.818,E2 -10709.818} C_VEL
LIN {X 0,Y 557.31,Z 511.078,A -85,B 0,C 180,E1 -10710.718,E2 -10710.718} C_VEL
LIN {X 0,Y 556.688,Z 521.555,A -85,B 0,C 180,E1 -10711.801,E2 -10711.801} C_VEL
LIN {X 0,Y 556.274,Z 530.193,A -85,B 0,C 180,E1 -10712.885,E2 -10712.885} C_VEL
LIN {X 0,Y 555.84,Z 537.406,A -85,B 0,C 180,E1 -10713.972,E2 -10713.972} C_VEL
LIN {X 0,Y 555.659,Z 544.198,A -85,B 0,C 180,E1 -10715.223,E2 -10715.223} C_VEL
LIN {X 0,Y 555.387,Z 549.796,A -85,B 0,C 180,E1 -10716.516,E2 -10716.516} C_VEL
LIN {X 0,Y 555.145,Z 554.589,A -85,B 0,C 180,E1 -10717.976,E2 -10717.976} C_VEL
LIN {X 0,Y 555.056,Z 557.892,A -85,B 0,C 180,E1 -10719.44,E2 -10719.44} C_VEL
LIN {X 0,Y 555.003,Z 559.791,A -85,B 0,C 180,E1 -10720.91,E2 -10720.91} C_VEL
LIN {X 0,Y 554.974,Z 560.34,A -85,B 0,C 180,E1 -10722.388,E2 -10722.388} C_VEL
LIN {X 0,Y 555.082,Z 559.529,A -85,B 0,C 180,E1 -10723.87,E2 -10723.87} C_VEL
LIN {X 0,Y 555.151,Z 557.336,A -85,B 0,C 180,E1 -10725.363,E2 -10725.363} C_VEL
LIN {X 0,Y 555.38,Z 553.675,A -85,B 0,C 180,E1 -10726.86,E2 -10726.86} C_VEL
LIN {X 0,Y 555.703,Z 548.424,A -85,B 0,C 180,E1 -10728.366,E2 -10728.366} C_VEL
LIN {X 0,Y 556.021,Z 543.26,A -85,B 0,C 180,E1 -10729.499,E2 -10729.499} C_VEL
LIN {X 0,Y 556.492,Z 535.811,A -85,B 0,C 180,E1 -10730.827,E2 -10730.827} C_VEL
LIN {X 0,Y 557.031,Z 527.916,A -85,B 0,C 180,E1 -10731.966,E2 -10731.966} C_VEL
LIN {X 0,Y 557.656,Z 518.469,A -85,B 0,C 180,E1 -10733.093,E2 -10733.093} C_VEL
LIN {X 0,Y 558.343,Z 507.552,A -85,B 0,C 180,E1 -10734.157,E2 -10734.157} C_VEL
LIN {X 0,Y 558.997,Z 496.886,A -85,B 0,C 180,E1 -10735.015,E2 -10735.015} C_VEL
LIN {X 0,Y 559.646,Z 483.918,A -85,B 0,C 180,E1 -10735.865,E2 -10735.865} C_VEL
LIN {X 0,Y 560.241,Z 470.706,A -85,B 0,C 180,E1 -10736.547,E2 -10736.547} C_VEL
LIN {X 0,Y 560.745,Z 457.411,A -85,B 0,C 180,E1 -10737.072,E2 -10737.072} C_VEL
LIN {X 0,Y 561.107,Z 442.957,A -85,B 0,C 180,E1 -10737.485,E2 -10737.485} C_VEL
LIN {X 0,Y 561.228,Z 428.847,A -85,B 0,C 180,E1 -10737.738,E2 -10737.738} C_VEL
LIN {X 0,Y 562.454,Z 318.959,A -85,B 0,C 180,E1 -10739.16,E2 -10739.16} C_VEL
LIN {X 0,Y 558.847,Z 302.954,A -85,B 0,C 180,E1 -10739.511,E2 -10739.511} C_VEL
LIN {X 0,Y 558.355,Z 300.94,A -85,B 0,C 180,E1 -10739.575,E2 -10739.575} C_VEL
LIN {X 0,Y 557.773,Z 295.812,A -85,B 0,C 180,E1 -10740.568,E2 -10740.568} C_VEL
LIN {X 0,Y 556.188,Z 287.765,A -85,B 0,C 180,E1 -10742.199,E2 -10742.199} C_VEL
LIN {X 0,Y 556.208,Z 287.758,A -85,B 0,C 180,E1 -10745.059,E2 -10745.059} C_VEL
LIN {X 0,Y 556.187,Z 287.76,A -85,B 0,C 180,E1 -10747.495,E2 -10747.495} C_VEL
LIN {X 0,Y 556.189,Z 287.757,A -85,B 0,C 180,E1 -10750.907,E2 -10750.907} C_VEL
LIN {X 0,Y 556.196,Z 287.762,A -85,B 0,C 180,E1 -10753.836,E2 -10753.836} C_VEL
LIN {X 0,Y 556.196,Z 287.762,A -85,B 0,C 180,E1 -10756.16,E2 -10756.16} C_VEL
LIN {X 0,Y 556.186,Z 287.759,A -85,B 0,C 180,E1 -10759.09,E2 -10759.09} C_VEL
LIN {X 0,Y 556.202,Z 287.762,A -85,B 0,C 180,E1 -10761.897,E2 -10761.897} C_VEL
LIN {X 0,Y 556.225,Z 287.74,A -85,B 0,C 180,E1 -10764.601,E2 -10764.601} C_VEL
LIN {X 0,Y 556.169,Z 287.766,A -85,B 0,C 180,E1 -10767.539,E2 -10767.539} C_VEL
LIN {X 0,Y 556.218,Z 287.755,A -85,B 0,C 180,E1 -10770.328,E2 -10770.328} C_VEL
LIN {X 0,Y 556.197,Z 287.752,A -85,B 0,C 180,E1 -10773.04,E2 -10773.04} C_VEL
LIN {X 0,Y 556.203,Z 287.763,A -85,B 0,C 180,E1 -10775.444,E2 -10775.444} C_VEL
LIN {X 0,Y 556.217,Z 287.759,A -85,B 0,C 180,E1 -10777.803,E2 -10777.803} C_VEL
LIN {X 0,Y 556.222,Z 287.751,A -85,B 0,C 180,E1 -10780.888,E2 -10780.888} C_VEL
LIN {X 0,Y 556.215,Z 287.755,A -85,B 0,C 180,E1 -10783.916,E2 -10783.916} C_VEL
LIN {X 0,Y 556.306,Z 287.737,A -85,B 0,C 180,E1 -10786.159,E2 -10786.159} C_VEL
LIN {X 0,Y 556.332,Z 287.746,A -85,B 0,C 180,E1 -10789.114,E2 -10789.114} C_VEL
LIN {X 0,Y 556.318,Z 287.739,A -85,B 0,C 180,E1 -10792.039,E2 -10792.039} C_VEL
LIN {X 0,Y 556.399,Z 287.736,A -85,B 0,C 180,E1 -10794.944,E2 -10794.944} C_VEL
LIN {X 0,Y 556.394,Z 287.732,A -85,B 0,C 180,E1 -10798.557,E2 -10798.557} C_VEL
LIN {X 0,Y 556.527,Z 287.714,A -85,B 0,C 180,E1 -10800,E2 -10800} C_VEL
LIN {X 0,Y 556.253,Z 287.74,A -85,B 0,C 180,E1 -10802.165,E2 -10802.165} C_VEL
LIN {X 0,Y 556.415,Z 287.735,A -85,B 0,C 180,E1 -10805.055,E2 -10805.055} C_VEL
LIN {X 0,Y 556.319,Z 287.733,A -85,B 0,C 180,E1 -10807.961,E2 -10807.961} C_VEL
LIN {X 0,Y 556.365,Z 287.738,A -85,B 0,C 180,E1 -10810.904,E2 -10810.904} C_VEL
LIN {X 0,Y 556.313,Z 287.739,A -85,B 0,C 180,E1 -10814.2,E2 -10814.2} C_VEL
LIN {X 0,Y 556.282,Z 287.743,A -85,B 0,C 180,E1 -10816.881,E2 -10816.881} C_VEL
LIN {X 0,Y 556.22,Z 287.752,A -85,B 0,C 180,E1 -10819.877,E2 -10819.877} C_VEL
LIN {X 0,Y 556.217,Z 287.75,A -85,B 0,C 180,E1 -10822.197,E2 -10822.197} C_VEL
LIN {X 0,Y 556.204,Z 287.757,A -85,B 0,C 180,E1 -10824.951,E2 -10824.951} C_VEL
LIN {X 0,Y 556.229,Z 287.755,A -85,B 0,C 180,E1 -10828.183,E2 -10828.183} C_VEL
LIN {X 0,Y 556.226,Z 287.753,A -85,B 0,C 180,E1 -10831.1,E2 -10831.1} C_VEL
LIN {X 0,Y 556.2,Z 287.755,A -85,B 0,C 180,E1 -10833.786,E2 -10833.786} C_VEL
LIN {X 0,Y 556.266,Z 287.735,A -85,B 0,C 180,E1 -10836.309,E2 -10836.309} C_VEL
LIN {X 0,Y 556.217,Z 287.755,A -85,B 0,C 180,E1 -10839.024,E2 -10839.024} C_VEL
LIN {X 0,Y 556.196,Z 287.762,A -85,B 0,C 180,E1 -10842.015,E2 -10842.015} C_VEL
LIN {X 0,Y 556.234,Z 287.749,A -85,B 0,C 180,E1 -10845.159,E2 -10845.159} C_VEL
LIN {X 0,Y 556.211,Z 287.761,A -85,B 0,C 180,E1 -10848.134,E2 -10848.134} C_VEL
LIN {X 0,Y 556.216,Z 287.754,A -85,B 0,C 180,E1 -10850.979,E2 -10850.979} C_VEL
LIN {X 0,Y 556.272,Z 287.748,A -85,B 0,C 180,E1 -10853.717,E2 -10853.717} C_VEL
LIN {X 0,Y 556.208,Z 287.759,A -85,B 0,C 180,E1 -10856.354,E2 -10856.354} C_VEL
LIN {X 0,Y 556.208,Z 287.763,A -85,B 0,C 180,E1 -10858.917,E2 -10858.917} C_VEL
LIN {X 0,Y 556.241,Z 287.759,A -85,B 0,C 180,E1 -10861.821,E2 -10861.821} C_VEL
LIN {X 0,Y 556.263,Z 287.874,A -85,B 0,C 180,E1 -10862.31,E2 -10862.31} C_VEL
LIN {X 0,Y 560.108,Z 305.616,A -85,B 0,C 180,E1 -10865.038,E2 -10865.038} C_VEL
LIN {X 0,Y 560.323,Z 309.844,A -85,B 0,C 180,E1 -10865.639,E2 -10865.639} C_VEL
LIN {X 0,Y 559.053,Z 329.598,A -85,B 0,C 180,E1 -10868.32,E2 -10868.32} C_VEL
LIN {X 0,Y 557.935,Z 350.696,A -85,B 0,C 180,E1 -10871.141,E2 -10871.141} C_VEL
LIN {X 0,Y 557.463,Z 360.582,A -85,B 0,C 180,E1 -10872.451,E2 -10872.451} C_VEL
LIN {X 0,Y 560.95,Z 383.477,A -85,B 0,C 180,E1 -10872.886,E2 -10872.886} C_VEL
LIN {X 0,Y 561.862,Z 392.647,A -85,B 0,C 180,E1 -10873.04,E2 -10873.04} C_VEL
LIN {X 0,Y 560.726,Z 499.26,A -85,B 0,C 180,E1 -10874.439,E2 -10874.439} C_VEL
LIN {X 0,Y 560.184,Z 513.917,A -85,B 0,C 180,E1 -10874.779,E2 -10874.779} C_VEL
LIN {X 0,Y 559.544,Z 528.273,A -85,B 0,C 180,E1 -10875.271,E2 -10875.271} C_VEL
LIN {X 0,Y 558.875,Z 541.046,A -85,B 0,C 180,E1 -10875.856,E2 -10875.856} C_VEL
LIN {X 0,Y 558.124,Z 553.502,A -85,B 0,C 180,E1 -10876.577,E2 -10876.577} C_VEL
LIN {X 0,Y 557.438,Z 564.903,A -85,B 0,C 180,E1 -10877.391,E2 -10877.391} C_VEL
LIN {X 0,Y 556.73,Z 576.384,A -85,B 0,C 180,E1 -10878.389,E2 -10878.389} C_VEL
LIN {X 0,Y 556.208,Z 586.978,A -85,B 0,C 180,E1 -10879.516,E2 -10879.516} C_VEL
LIN {X 0,Y 555.732,Z 595.223,A -85,B 0,C 180,E1 -10880.571,E2 -10880.571} C_VEL
LIN {X 0,Y 555.289,Z 603.414,A -85,B 0,C 180,E1 -10881.844,E2 -10881.844} C_VEL
LIN {X 0,Y 555.05,Z 612.252,A -85,B 0,C 180,E1 -10883.48,E2 -10883.48} C_VEL
LIN {X 0,Y 554.975,Z 617.093,A -85,B 0,C 180,E1 -10884.57,E2 -10884.57} C_VEL
LIN {X 0,Y 554.925,Z 621.05,A -85,B 0,C 180,E1 -10885.685,E2 -10885.685} C_VEL
LIN {X 0,Y 554.917,Z 624.717,A -85,B 0,C 180,E1 -10887.108,E2 -10887.108} C_VEL
LIN {X 0,Y 554.875,Z 626.985,A -85,B 0,C 180,E1 -10888.555,E2 -10888.555} C_VEL
LIN {X 0,Y 554.892,Z 627.83,A -85,B 0,C 180,E1 -10890.002,E2 -10890.002} C_VEL
LIN {X 0,Y 554.875,Z 627.261,A -85,B 0,C 180,E1 -10891.448,E2 -10891.448} C_VEL
LIN {X 0,Y 554.92,Z 625.264,A -85,B 0,C 180,E1 -10892.896,E2 -10892.896} C_VEL
LIN {X 0,Y 554.909,Z 621.774,A -85,B 0,C 180,E1 -10894.345,E2 -10894.345} C_VEL
LIN {X 0,Y 554.981,Z 618.164,A -85,B 0,C 180,E1 -10895.433,E2 -10895.433} C_VEL
LIN {X 0,Y 555.068,Z 613.561,A -85,B 0,C 180,E1 -10896.523,E2 -10896.523} C_VEL
LIN {X 0,Y 555.29,Z 606.915,A -85,B 0,C 180,E1 -10897.795,E2 -10897.795} C_VEL
LIN {X 0,Y 555.641,Z 598.639,A -85,B 0,C 180,E1 -10899.068,E2 -10899.068} C_VEL
LIN {X 0,Y 555.961,Z 589.949,A -85,B 0,C 180,E1 -10900.161,E2 -10900.161} C_VEL
LIN {X 0,Y 556.459,Z 581.321,A -85,B 0,C 180,E1 -10901.069,E2 -10901.069} C_VEL
LIN {X 0,Y 556.94,Z 569.954,A -85,B 0,C 180,E1 -10902.07,E2 -10902.07} C_VEL
LIN {X 0,Y 557.463,Z 558.67,A -85,B 0,C 180,E1 -10902.888,E2 -10902.888} C_VEL
LIN {X 0,Y 558.091,Z 546.387,A -85,B 0,C 180,E1 -10903.612,E2 -10903.612} C_VEL
LIN {X 0,Y 558.682,Z 532.804,A -85,B 0,C 180,E1 -10904.245,E2 -10904.245} C_VEL
LIN {X 0,Y 559.129,Z 518.683,A -85,B 0,C 180,E1 -10904.743,E2 -10904.743} C_VEL
LIN {X 0,Y 559.597,Z 504.96,A -85,B 0,C 180,E1 -10905.079,E2 -10905.079} C_VEL
LIN {X 0,Y 561.384,Z 389.945,A -85,B 0,C 180,E1 -10906.859,E2 -10906.859} C_VEL
LIN {X 0,Y 558.411,Z 365.196,A -85,B 0,C 180,E1 -10907.391,E2 -10907.391} C_VEL
LIN {X 0,Y 557.131,Z 356.562,A -85,B 0,C 180,E1 -10907.611,E2 -10907.611} C_VEL
LIN {X 0,Y 558.028,Z 335.216,A -85,B 0,C 180,E1 -10910.386,E2 -10910.386} C_VEL
LIN {X 0,Y 559.157,Z 311.967,A -85,B 0,C 180,E1 -10913.438,E2 -10913.438} C_VEL
LIN {X 0,Y 559.482,Z 304.673,A -85,B 0,C 180,E1 -10914.404,E2 -10914.404} C_VEL
LIN {X 0,Y 556.455,Z 288.902,A -85,B 0,C 180,E1 -10916.655,E2 -10916.655} C_VEL
LIN {X 0,Y 556.246,Z 287.756,A -85,B 0,C 180,E1 -10916.858,E2 -10916.858} C_VEL
LIN {X 0,Y 556.225,Z 287.759,A -85,B 0,C 180,E1 -10919.668,E2 -10919.668} C_VEL
LIN {X 0,Y 556.194,Z 287.757,A -85,B 0,C 180,E1 -10922.46,E2 -10922.46} C_VEL
LIN {X 0,Y 556.195,Z 287.763,A -85,B 0,C 180,E1 -10925.403,E2 -10925.403} C_VEL
LIN {X 0,Y 556.178,Z 287.762,A -85,B 0,C 180,E1 -10928.106,E2 -10928.106} C_VEL
LIN {X 0,Y 556.202,Z 287.76,A -85,B 0,C 180,E1 -10930.922,E2 -10930.922} C_VEL
LIN {X 0,Y 556.209,Z 287.755,A -85,B 0,C 180,E1 -10934.126,E2 -10934.126} C_VEL
LIN {X 0,Y 556.183,Z 287.763,A -85,B 0,C 180,E1 -10936.925,E2 -10936.925} C_VEL
LIN {X 0,Y 556.212,Z 287.762,A -85,B 0,C 180,E1 -10939.092,E2 -10939.092} C_VEL
LIN {X 0,Y 556.207,Z 287.761,A -85,B 0,C 180,E1 -10942.504,E2 -10942.504} C_VEL
LIN {X 0,Y 556.24,Z 287.758,A -85,B 0,C 180,E1 -10944.938,E2 -10944.938} C_VEL
LIN {X 0,Y 556.212,Z 287.758,A -85,B 0,C 180,E1 -10948.068,E2 -10948.068} C_VEL
LIN {X 0,Y 556.229,Z 287.76,A -85,B 0,C 180,E1 -10950.586,E2 -10950.586} C_VEL
LIN {X 0,Y 556.225,Z 287.756,A -85,B 0,C 180,E1 -10953.394,E2 -10953.394} C_VEL
LIN {X 0,Y 556.227,Z 287.762,A -85,B 0,C 180,E1 -10956.236,E2 -10956.236} C_VEL
LIN {X 0,Y 556.265,Z 287.758,A -85,B 0,C 180,E1 -10958.72,E2 -10958.72} C_VEL
LIN {X 0,Y 556.244,Z 287.76,A -85,B 0,C 180,E1 -10961.651,E2 -10961.651} C_VEL
LIN {X 0,Y 556.267,Z 287.753,A -85,B 0,C 180,E1 -10964.667,E2 -10964.667} C_VEL
LIN {X 0,Y 556.303,Z 287.912,A -85,B 0,C 180,E1 -10967.016,E2 -10967.016} C_VEL
LIN {X 0,Y 559.358,Z 301.672,A -85,B 0,C 180,E1 -10968.991,E2 -10968.991} C_VEL
LIN {X 0,Y 559.724,Z 305.72,A -85,B 0,C 180,E1 -10969.545,E2 -10969.545} C_VEL
LIN {X 0,Y 559.228,Z 325.255,A -85,B 0,C 180,E1 -10972.081,E2 -10972.081} C_VEL
LIN {X 0,Y 558.594,Z 343.659,A -85,B 0,C 180,E1 -10974.457,E2 -10974.457} C_VEL
LIN {X 0,Y 561.794,Z 360.464,A -85,B 0,C 180,E1 -10974.87,E2 -10974.87} C_VEL
LIN {X 0,Y 562.306,Z 364.245,A -85,B 0,C 180,E1 -10974.953,E2 -10974.953} C_VEL
LIN {X 0,Y 560.237,Z 482.544,A -85,B 0,C 180,E1 -10976.775,E2 -10976.775} C_VEL
LIN {X 0,Y 559.854,Z 496.697,A -85,B 0,C 180,E1 -10977.131,E2 -10977.131} C_VEL
LIN {X 0,Y 559.302,Z 510.434,A -85,B 0,C 180,E1 -10977.622,E2 -10977.622} C_VEL
LIN {X 0,Y 558.79,Z 522.869,A -85,B 0,C 180,E1 -10978.204,E2 -10978.204} C_VEL
LIN {X 0,Y 558.155,Z 535.131,A -85,B 0,C 180,E1 -10978.921,E2 -10978.921} C_VEL
LIN {X 0,Y 557.579,Z 547.506,A -85,B 0,C 180,E1 -10979.82,E2 -10979.82} C_VEL
LIN {X 0,Y 557.058,Z 557.731,A -85,B 0,C 180,E1 -10980.72,E2 -10980.72} C_VEL
LIN {X 0,Y 556.362,Z 567.994,A -85,B 0,C 180,E1 -10981.804,E2 -10981.804} C_VEL
LIN {X 0,Y 555.984,Z 576.464,A -85,B 0,C 180,E1 -10982.889,E2 -10982.889} C_VEL
LIN {X 0,Y 555.508,Z 583.549,A -85,B 0,C 180,E1 -10983.977,E2 -10983.977} C_VEL
LIN {X 0,Y 555.401,Z 589.39,A -85,B 0,C 180,E1 -10985.065,E2 -10985.065} C_VEL
LIN {X 0,Y 555.203,Z 594.227,A -85,B 0,C 180,E1 -10986.156,E2 -10986.156} C_VEL
LIN {X 0,Y 554.967,Z 599.212,A -85,B 0,C 180,E1 -10987.615,E2 -10987.615} C_VEL
LIN {X 0,Y 554.887,Z 601.932,A -85,B 0,C 180,E1 -10988.713,E2 -10988.713} C_VEL
LIN {X 0,Y 554.883,Z 604.259,A -85,B 0,C 180,E1 -10990.179,E2 -10990.179} C_VEL
LIN {X 0,Y 554.746,Z 605.17,A -85,B 0,C 180,E1 -10991.655,E2 -10991.655} C_VEL
LIN {X 0,Y 554.832,Z 604.642,A -85,B 0,C 180,E1 -10993.135,E2 -10993.135} C_VEL
LIN {X 0,Y 554.788,Z 602.634,A -85,B 0,C 180,E1 -10994.626,E2 -10994.626} C_VEL
LIN {X 0,Y 554.93,Z 599.059,A -85,B 0,C 180,E1 -10996.122,E2 -10996.122} C_VEL
LIN {X 0,Y 555,Z 595.316,A -85,B 0,C 180,E1 -10997.253,E2 -10997.253} C_VEL
LIN {X 0,Y 555.218,Z 589.295,A -85,B 0,C 180,E1 -10998.637,E2 -10998.637} C_VEL
LIN {X 0,Y 555.474,Z 582.295,A -85,B 0,C 180,E1 -10999.905,E2 -10999.905} C_VEL
LIN {X 0,Y 555.851,Z 573.641,A -85,B 0,C 180,E1 -11001.17,E2 -11001.17} C_VEL
LIN {X 0,Y 556.171,Z 565.101,A -85,B 0,C 180,E1 -11002.199,E2 -11002.199} C_VEL
LIN {X 0,Y 556.677,Z 554.24,A -85,B 0,C 180,E1 -11003.286,E2 -11003.286} C_VEL
LIN {X 0,Y 557.198,Z 542.899,A -85,B 0,C 180,E1 -11004.213,E2 -11004.213} C_VEL
LIN {X 0,Y 557.697,Z 529.853,A -85,B 0,C 180,E1 -11005.08,E2 -11005.08} C_VEL
LIN {X 0,Y 558.24,Z 516.227,A -85,B 0,C 180,E1 -11005.8,E2 -11005.8} C_VEL
LIN {X 0,Y 558.714,Z 501.98,A -85,B 0,C 180,E1 -11006.377,E2 -11006.377} C_VEL
LIN {X 0,Y 559.185,Z 488.155,A -85,B 0,C 180,E1 -11006.779,E2 -11006.779} C_VEL
LIN {X 0,Y 559.393,Z 472.466,A -85,B 0,C 180,E1 -11007.078,E2 -11007.078} C_VEL
LIN {X 0,Y 560.746,Z 362.528,A -85,B 0,C 180,E1 -11008.666,E2 -11008.666} C_VEL
LIN {X 0,Y 557.634,Z 342.337,A -85,B 0,C 180,E1 -11009.066,E2 -11009.066} C_VEL
LIN {X 0,Y 558.34,Z 320.116,A -85,B 0,C 180,E1 -11012.008,E2 -11012.008} C_VEL
LIN {X 0,Y 558.89,Z 302.56,A -85,B 0,C 180,E1 -11014.331,E2 -11014.331} C_VEL
LIN {X 0,Y 556.783,Z 290.363,A -85,B 0,C 180,E1 -11016.024,E2 -11016.024} C_VEL
LIN {X 0,Y 556.253,Z 287.757,A -85,B 0,C 180,E1 -11016.418,E2 -11016.418} C_VEL
LIN {X 0,Y 556.196,Z 287.758,A -85,B 0,C 180,E1 -11019.026,E2 -11019.026} C_VEL
LIN {X 0,Y 556.205,Z 287.76,A -85,B 0,C 180,E1 -11022.011,E2 -11022.011} C_VEL
LIN {X 0,Y 556.256,Z 287.751,A -85,B 0,C 180,E1 -11025.156,E2 -11025.156} C_VEL
LIN {X 0,Y 556.166,Z 287.767,A -85,B 0,C 180,E1 -11028.125,E2 -11028.125} C_VEL
LIN {X 0,Y 556.185,Z 287.763,A -85,B 0,C 180,E1 -11030.194,E2 -11030.194} C_VEL
LIN {X 0,Y 556.166,Z 287.765,A -85,B 0,C 180,E1 -11032.804,E2 -11032.804} C_VEL
LIN {X 0,Y 556.208,Z 287.759,A -85,B 0,C 180,E1 -11035.478,E2 -11035.478} C_VEL
LIN {X 0,Y 556.207,Z 287.759,A -85,B 0,C 180,E1 -11038.066,E2 -11038.066} C_VEL
LIN {X 0,Y 556.225,Z 287.759,A -85,B 0,C 180,E1 -11040.584,E2 -11040.584} C_VEL
LIN {X 0,Y 556.223,Z 287.757,A -85,B 0,C 180,E1 -11043.392,E2 -11043.392} C_VEL
LIN {X 0,Y 556.225,Z 287.758,A -85,B 0,C 180,E1 -11046.234,E2 -11046.234} C_VEL
LIN {X 0,Y 556.237,Z 287.754,A -85,B 0,C 180,E1 -11048.351,E2 -11048.351} C_VEL
LIN {X 0,Y 555.592,Z 287.836,A -85,B 0,C 180,E1 -11048.955,E2 -11048.955} C_VEL
LIN {X 0,Y 552.745,Z 288.191,A -85,B 0,C 180,E1 -11049.935,E2 -11049.935} C_VEL
LIN {X 0,Y 550.323,Z 288.492,A -85,B 0,C 180,E1 -11050.724,E2 -11050.724} C_VEL
LIN {X 0,Y 549.279,Z 288.621,A -85,B 0,C 180,E1 -11051.334,E2 -11051.334} C_VEL
LIN {X 0,Y 549.192,Z 288.632,A -85,B 0,C 180,E1 -11051.54,E2 -11051.54} C_VEL
LIN {X 0,Y 549.237,Z 288.627,A -85,B 0,C 180,E1 -11053.704,E2 -11053.704} C_VEL
LIN {X 0,Y 549.287,Z 288.624,A -85,B 0,C 180,E1 -11055.977,E2 -11055.977} C_VEL
LIN {X 0,Y 549.328,Z 288.613,A -85,B 0,C 180,E1 -11059.059,E2 -11059.059} C_VEL
LIN {X 0,Y 549.346,Z 288.616,A -85,B 0,C 180,E1 -11062.489,E2 -11062.489} C_VEL
LIN {X 0,Y 549.349,Z 288.743,A -85,B 0,C 180,E1 -11062.627,E2 -11062.627} C_VEL
LIN {X 0,Y 550.582,Z 296.796,A -85,B 0,C 180,E1 -11064.157,E2 -11064.157} C_VEL
LIN {X 0,Y 550.482,Z 301.129,A -85,B 0,C 180,E1 -11064.902,E2 -11064.902} C_VEL
LIN {X 0,Y 554.149,Z 319.022,A -85,B 0,C 180,E1 -11065.24,E2 -11065.24} C_VEL
LIN {X 0,Y 552.991,Z 436.427,A -85,B 0,C 180,E1 -11066.776,E2 -11066.776} C_VEL
LIN {X 0,Y 552.66,Z 450.878,A -85,B 0,C 180,E1 -11067.115,E2 -11067.115} C_VEL
LIN {X 0,Y 552.317,Z 464.661,A -85,B 0,C 180,E1 -11067.591,E2 -11067.591} C_VEL
LIN {X 0,Y 551.895,Z 477.503,A -85,B 0,C 180,E1 -11068.18,E2 -11068.18} C_VEL
LIN {X 0,Y 551.432,Z 489.962,A -85,B 0,C 180,E1 -11068.906,E2 -11068.906} C_VEL
LIN {X 0,Y 550.723,Z 501.406,A -85,B 0,C 180,E1 -11069.725,E2 -11069.725} C_VEL
LIN {X 0,Y 550.25,Z 512.803,A -85,B 0,C 180,E1 -11070.728,E2 -11070.728} C_VEL
LIN {X 0,Y 549.61,Z 523.063,A -85,B 0,C 180,E1 -11071.824,E2 -11071.824} C_VEL
LIN {X 0,Y 549.225,Z 531.513,A -85,B 0,C 180,E1 -11072.922,E2 -11072.922} C_VEL
LIN {X 0,Y 548.7,Z 539.639,A -85,B 0,C 180,E1 -11074.208,E2 -11074.208} C_VEL
LIN {X 0,Y 548.544,Z 546.156,A -85,B 0,C 180,E1 -11075.493,E2 -11075.493} C_VEL
LIN {X 0,Y 548.267,Z 551.976,A -85,B 0,C 180,E1 -11076.969,E2 -11076.969} C_VEL
LIN {X 0,Y 548.047,Z 555.351,A -85,B 0,C 180,E1 -11078.08,E2 -11078.08} C_VEL
LIN {X 0,Y 547.978,Z 558.504,A -85,B 0,C 180,E1 -11079.563,E2 -11079.563} C_VEL
LIN {X 0,Y 547.914,Z 560.29,A -85,B 0,C 180,E1 -11081.053,E2 -11081.053} C_VEL
LIN {X 0,Y 547.915,Z 560.728,A -85,B 0,C 180,E1 -11082.55,E2 -11082.55} C_VEL
LIN {X 0,Y 548.021,Z 559.808,A -85,B 0,C 180,E1 -11084.052,E2 -11084.052} C_VEL
LIN {X 0,Y 548.094,Z 557.501,A -85,B 0,C 180,E1 -11085.565,E2 -11085.565} C_VEL
LIN {X 0,Y 548.333,Z 553.722,A -85,B 0,C 180,E1 -11087.084,E2 -11087.084} C_VEL
LIN {X 0,Y 548.605,Z 549.794,A -85,B 0,C 180,E1 -11088.226,E2 -11088.226} C_VEL
LIN {X 0,Y 548.954,Z 544.892,A -85,B 0,C 180,E1 -11089.373,E2 -11089.373} C_VEL
LIN {X 0,Y 549.383,Z 537.733,A -85,B 0,C 180,E1 -11090.718,E2 -11090.718} C_VEL
LIN {X 0,Y 549.947,Z 530.168,A -85,B 0,C 180,E1 -11091.87,E2 -11091.87} C_VEL
LIN {X 0,Y 550.597,Z 520.979,A -85,B 0,C 180,E1 -11093.026,E2 -11093.026} C_VEL
LIN {X 0,Y 551.3,Z 510.746,A -85,B 0,C 180,E1 -11094.087,E2 -11094.087} C_VEL
LIN {X 0,Y 552.066,Z 499.43,A -85,B 0,C 180,E1 -11095.05,E2 -11095.05} C_VEL
LIN {X 0,Y 552.694,Z 487.709,A -85,B 0,C 180,E1 -11095.868,E2 -11095.868} C_VEL
LIN {X 0,Y 553.32,Z 474.544,A -85,B 0,C 180,E1 -11096.601,E2 -11096.601} C_VEL
LIN {X 0,Y 553.84,Z 461.075,A -85,B 0,C 180,E1 -11097.178,E2 -11097.178} C_VEL
LIN {X 0,Y 554.205,Z 447.129,A -85,B 0,C 180,E1 -11097.617,E2 -11097.617} C_VEL
LIN {X 0,Y 554.515,Z 432.689,A -85,B 0,C 180,E1 -11097.912,E2 -11097.912} C_VEL
LIN {X 0,Y 555.705,Z 319.219,A -85,B 0,C 180,E1 -11099.411,E2 -11099.411} C_VEL
LIN {X 0,Y 551.424,Z 301.443,A -85,B 0,C 180,E1 -11099.827,E2 -11099.827} C_VEL
LIN {X 0,Y 550.075,Z 293.31,A -85,B 0,C 180,E1 -11101.444,E2 -11101.444} C_VEL
LIN {X 0,Y 549.162,Z 288.642,A -85,B 0,C 180,E1 -11102.423,E2 -11102.423} C_VEL
LIN {X 0,Y 549.162,Z 288.636,A -85,B 0,C 180,E1 -11105.283,E2 -11105.283} C_VEL
LIN {X 0,Y 549.15,Z 288.64,A -85,B 0,C 180,E1 -11107.749,E2 -11107.749} C_VEL
LIN {X 0,Y 549.136,Z 288.638,A -85,B 0,C 180,E1 -11110.578,E2 -11110.578} C_VEL
LIN {X 0,Y 549.164,Z 288.638,A -85,B 0,C 180,E1 -11113.528,E2 -11113.528} C_VEL
LIN {X 0,Y 549.163,Z 288.636,A -85,B 0,C 180,E1 -11116.468,E2 -11116.468} C_VEL
LIN {X 0,Y 549.139,Z 288.639,A -85,B 0,C 180,E1 -11119.419,E2 -11119.419} C_VEL
LIN {X 0,Y 549.152,Z 288.634,A -85,B 0,C 180,E1 -11122.257,E2 -11122.257} C_VEL
LIN {X 0,Y 549.169,Z 288.619,A -85,B 0,C 180,E1 -11124.973,E2 -11124.973} C_VEL
LIN {X 0,Y 549.124,Z 288.644,A -85,B 0,C 180,E1 -11127.606,E2 -11127.606} C_VEL
LIN {X 0,Y 549.168,Z 288.635,A -85,B 0,C 180,E1 -11130.17,E2 -11130.17} C_VEL
LIN {X 0,Y 549.171,Z 288.626,A -85,B 0,C 180,E1 -11132.667,E2 -11132.667} C_VEL
LIN {X 0,Y 549.156,Z 288.632,A -85,B 0,C 180,E1 -11135.911,E2 -11135.911} C_VEL
LIN {X 0,Y 549.186,Z 288.629,A -85,B 0,C 180,E1 -11138.593,E2 -11138.593} C_VEL
LIN {X 0,Y 549.162,Z 288.632,A -85,B 0,C 180,E1 -11141.405,E2 -11141.405} C_VEL
LIN {X 0,Y 549.199,Z 288.627,A -85,B 0,C 180,E1 -11144.465,E2 -11144.465} C_VEL
LIN {X 0,Y 549.218,Z 288.62,A -85,B 0,C 180,E1 -11146.729,E2 -11146.729} C_VEL
LIN {X 0,Y 549.271,Z 288.618,A -85,B 0,C 180,E1 -11149.716,E2 -11149.716} C_VEL
LIN {X 0,Y 549.312,Z 288.612,A -85,B 0,C 180,E1 -11152.674,E2 -11152.674} C_VEL
LIN {X 0,Y 549.353,Z 288.603,A -85,B 0,C 180,E1 -11155.612,E2 -11155.612} C_VEL
LIN {X 0,Y 549.51,Z 288.595,A -85,B 0,C 180,E1 -11159.27,E2 -11159.27} C_VEL
LIN {X 0,Y 549.376,Z 288.599,A -85,B 0,C 180,E1 -11161.461,E2 -11161.461} C_VEL
LIN {X 0,Y 549.361,Z 288.608,A -85,B 0,C 180,E1 -11164.387,E2 -11164.387} C_VEL
LIN {X 0,Y 549.307,Z 288.615,A -85,B 0,C 180,E1 -11166.59,E2 -11166.59} C_VEL
LIN {X 0,Y 549.232,Z 288.624,A -85,B 0,C 180,E1 -11169.543,E2 -11169.543} C_VEL
LIN {X 0,Y 549.254,Z 288.614,A -85,B 0,C 180,E1 -11171.773,E2 -11171.773} C_VEL
LIN {X 0,Y 549.245,Z 288.627,A -85,B 0,C 180,E1 -11174.777,E2 -11174.777} C_VEL
LIN {X 0,Y 549.195,Z 288.619,A -85,B 0,C 180,E1 -11177.824,E2 -11177.824} C_VEL
LIN {X 0,Y 549.186,Z 288.63,A -85,B 0,C 180,E1 -11180.923,E2 -11180.923} C_VEL
LIN {X 0,Y 549.157,Z 288.633,A -85,B 0,C 180,E1 -11183.32,E2 -11183.32} C_VEL
LIN {X 0,Y 549.111,Z 288.636,A -85,B 0,C 180,E1 -11185.703,E2 -11185.703} C_VEL
LIN {X 0,Y 549.176,Z 288.636,A -85,B 0,C 180,E1 -11188.356,E2 -11188.356} C_VEL
LIN {X 0,Y 549.172,Z 288.631,A -85,B 0,C 180,E1 -11191.294,E2 -11191.294} C_VEL
LIN {X 0,Y 549.173,Z 288.63,A -85,B 0,C 180,E1 -11194.139,E2 -11194.139} C_VEL
LIN {X 0,Y 549.205,Z 288.623,A -85,B 0,C 180,E1 -11196.829,E2 -11196.829} C_VEL
LIN {X 0,Y 549.18,Z 288.631,A -85,B 0,C 180,E1 -11199.622,E2 -11199.622} C_VEL
LIN {X 0,Y 549.166,Z 288.635,A -85,B 0,C 180,E1 -11202.532,E2 -11202.532} C_VEL
LIN {X 0,Y 549.182,Z 288.629,A -85,B 0,C 180,E1 -11205.581,E2 -11205.581} C_VEL
LIN {X 0,Y 549.173,Z 288.636,A -85,B 0,C 180,E1 -11208.456,E2 -11208.456} C_VEL
LIN {X 0,Y 549.184,Z 288.631,A -85,B 0,C 180,E1 -11211.324,E2 -11211.324} C_VEL
LIN {X 0,Y 549.226,Z 288.628,A -85,B 0,C 180,E1 -11214.083,E2 -11214.083} C_VEL
LIN {X 0,Y 549.156,Z 288.639,A -85,B 0,C 180,E1 -11216.741,E2 -11216.741} C_VEL
LIN {X 0,Y 549.172,Z 288.64,A -85,B 0,C 180,E1 -11219.327,E2 -11219.327} C_VEL
LIN {X 0,Y 549.217,Z 288.713,A -85,B 0,C 180,E1 -11222.053,E2 -11222.053} C_VEL
LIN {X 0,Y 552.916,Z 305.523,A -85,B 0,C 180,E1 -11224.69,E2 -11224.69} C_VEL
LIN {X 0,Y 553.5,Z 309.756,A -85,B 0,C 180,E1 -11225.319,E2 -11225.319} C_VEL
LIN {X 0,Y 552.215,Z 329.888,A -85,B 0,C 180,E1 -11228.097,E2 -11228.097} C_VEL
LIN {X 0,Y 550.95,Z 351.939,A -85,B 0,C 180,E1 -11231.086,E2 -11231.086} C_VEL
LIN {X 0,Y 550.571,Z 360.282,A -85,B 0,C 180,E1 -11232.191,E2 -11232.191} C_VEL
LIN {X 0,Y 554.229,Z 383.95,A -85,B 0,C 180,E1 -11232.65,E2 -11232.65} C_VEL
LIN {X 0,Y 555.159,Z 393.504,A -85,B 0,C 180,E1 -11232.813,E2 -11232.813} C_VEL
LIN {X 0,Y 553.993,Z 498.329,A -85,B 0,C 180,E1 -11234.202,E2 -11234.202} C_VEL
LIN {X 0,Y 553.458,Z 512.84,A -85,B 0,C 180,E1 -11234.537,E2 -11234.537} C_VEL
LIN {X 0,Y 552.818,Z 526.368,A -85,B 0,C 180,E1 -11234.994,E2 -11234.994} C_VEL
LIN {X 0,Y 552.135,Z 539.456,A -85,B 0,C 180,E1 -11235.586,E2 -11235.586} C_VEL
LIN {X 0,Y 551.321,Z 552.13,A -85,B 0,C 180,E1 -11236.314,E2 -11236.314} C_VEL
LIN {X 0,Y 550.552,Z 563.693,A -85,B 0,C 180,E1 -11237.138,E2 -11237.138} C_VEL
LIN {X 0,Y 549.84,Z 574.327,A -85,B 0,C 180,E1 -11238.055,E2 -11238.055} C_VEL
LIN {X 0,Y 549.347,Z 583.918,A -85,B 0,C 180,E1 -11239.049,E2 -11239.049} C_VEL
LIN {X 0,Y 548.749,Z 593.664,A -85,B 0,C 180,E1 -11240.265,E2 -11240.265} C_VEL
LIN {X 0,Y 548.262,Z 602.094,A -85,B 0,C 180,E1 -11241.553,E2 -11241.553} C_VEL
LIN {X 0,Y 547.972,Z 611.897,A -85,B 0,C 180,E1 -11243.396,E2 -11243.396} C_VEL
LIN {X 0,Y 547.876,Z 616.785,A -85,B 0,C 180,E1 -11244.5,E2 -11244.5} C_VEL
LIN {X 0,Y 547.846,Z 621.18,A -85,B 0,C 180,E1 -11245.761,E2 -11245.761} C_VEL
LIN {X 0,Y 547.829,Z 624.495,A -85,B 0,C 180,E1 -11247.07,E2 -11247.07} C_VEL
LIN {X 0,Y 547.793,Z 626.798,A -85,B 0,C 180,E1 -11248.536,E2 -11248.536} C_VEL
LIN {X 0,Y 547.802,Z 627.673,A -85,B 0,C 180,E1 -11250.002,E2 -11250.002} C_VEL
LIN {X 0,Y 547.792,Z 627.13,A -85,B 0,C 180,E1 -11251.467,E2 -11251.467} C_VEL
LIN {X 0,Y 547.832,Z 625.163,A -85,B 0,C 180,E1 -11252.933,E2 -11252.933} C_VEL
LIN {X 0,Y 547.822,Z 621.7,A -85,B 0,C 180,E1 -11254.402,E2 -11254.402} C_VEL
LIN {X 0,Y 547.9,Z 618.102,A -85,B 0,C 180,E1 -11255.504,E2 -11255.504} C_VEL
LIN {X 0,Y 547.997,Z 613.527,A -85,B 0,C 180,E1 -11256.607,E2 -11256.607} C_VEL
LIN {X 0,Y 548.213,Z 606.898,A -85,B 0,C 180,E1 -11257.896,E2 -11257.896} C_VEL
LIN {X 0,Y 548.62,Z 598.647,A -85,B 0,C 180,E1 -11259.185,E2 -11259.185} C_VEL
LIN {X 0,Y 548.968,Z 589.999,A -85,B 0,C 180,E1 -11260.292,E2 -11260.292} C_VEL
LIN {X 0,Y 549.538,Z 579.504,A -85,B 0,C 180,E1 -11261.396,E2 -11261.396} C_VEL
LIN {X 0,Y 550.073,Z 567.771,A -85,B 0,C 180,E1 -11262.41,E2 -11262.41} C_VEL
LIN {X 0,Y 550.739,Z 556.059,A -85,B 0,C 180,E1 -11263.236,E2 -11263.236} C_VEL
LIN {X 0,Y 551.342,Z 543.217,A -85,B 0,C 180,E1 -11263.97,E2 -11263.97} C_VEL
LIN {X 0,Y 551.998,Z 529.983,A -85,B 0,C 180,E1 -11264.562,E2 -11264.562} C_VEL
LIN {X 0,Y 552.463,Z 517.252,A -85,B 0,C 180,E1 -11264.996,E2 -11264.996} C_VEL
LIN {X 0,Y 552.859,Z 502.841,A -85,B 0,C 180,E1 -11265.337,E2 -11265.337} C_VEL
LIN {X 0,Y 554.812,Z 391.684,A -85,B 0,C 180,E1 -11267.086,E2 -11267.086} C_VEL
LIN {X 0,Y 551.86,Z 366.376,A -85,B 0,C 180,E1 -11267.642,E2 -11267.642} C_VEL
LIN {X 0,Y 550.149,Z 355.357,A -85,B 0,C 180,E1 -11267.914,E2 -11267.914} C_VEL
LIN {X 0,Y 551.022,Z 336.017,A -85,B 0,C 180,E1 -11270.463,E2 -11270.463} C_VEL
LIN {X 0,Y 552.139,Z 314.21,A -85,B 0,C 180,E1 -11273.357,E2 -11273.357} C_VEL
LIN {X 0,Y 552.478,Z 305.396,A -85,B 0,C 180,E1 -11274.544,E2 -11274.544} C_VEL
LIN {X 0,Y 549.225,Z 288.63,A -85,B 0,C 180,E1 -11276.982,E2 -11276.982} C_VEL
LIN {X 0,Y 549.173,Z 288.635,A -85,B 0,C 180,E1 -11279.853,E2 -11279.853} C_VEL
LIN {X 0,Y 549.149,Z 288.634,A -85,B 0,C 180,E1 -11282.665,E2 -11282.665} C_VEL
LIN {X 0,Y 549.176,Z 288.638,A -85,B 0,C 180,E1 -11285.285,E2 -11285.285} C_VEL
LIN {X 0,Y 549.148,Z 288.64,A -85,B 0,C 180,E1 -11287.754,E2 -11287.754} C_VEL
LIN {X 0,Y 549.158,Z 288.635,A -85,B 0,C 180,E1 -11290.581,E2 -11290.581} C_VEL
LIN {X 0,Y 549.134,Z 288.64,A -85,B 0,C 180,E1 -11293.536,E2 -11293.536} C_VEL
LIN {X 0,Y 549.191,Z 288.633,A -85,B 0,C 180,E1 -11295.582,E2 -11295.582} C_VEL
LIN {X 0,Y 549.155,Z 288.638,A -85,B 0,C 180,E1 -11298.813,E2 -11298.813} C_VEL
LIN {X 0,Y 549.135,Z 288.641,A -85,B 0,C 180,E1 -11301.317,E2 -11301.317} C_VEL
LIN {X 0,Y 549.2,Z 288.631,A -85,B 0,C 180,E1 -11304.078,E2 -11304.078} C_VEL
LIN {X 0,Y 549.134,Z 288.643,A -85,B 0,C 180,E1 -11306.737,E2 -11306.737} C_VEL
LIN {X 0,Y 549.18,Z 288.633,A -85,B 0,C 180,E1 -11309.324,E2 -11309.324} C_VEL
LIN {X 0,Y 549.201,Z 288.63,A -85,B 0,C 180,E1 -11311.843,E2 -11311.843} C_VEL
LIN {X 0,Y 549.179,Z 288.636,A -85,B 0,C 180,E1 -11314.901,E2 -11314.901} C_VEL
LIN {X 0,Y 549.204,Z 288.634,A -85,B 0,C 180,E1 -11317.504,E2 -11317.504} C_VEL
LIN {X 0,Y 549.202,Z 288.642,A -85,B 0,C 180,E1 -11319.858,E2 -11319.858} C_VEL
LIN {X 0,Y 549.194,Z 288.633,A -85,B 0,C 180,E1 -11322.942,E2 -11322.942} C_VEL
LIN {X 0,Y 549.276,Z 288.626,A -85,B 0,C 180,E1 -11325.978,E2 -11325.978} C_VEL
LIN {X 0,Y 549.238,Z 288.727,A -85,B 0,C 180,E1 -11326.729,E2 -11326.729} C_VEL
LIN {X 0,Y 552.298,Z 302.019,A -85,B 0,C 180,E1 -11328.663,E2 -11328.663} C_VEL
LIN {X 0,Y 552.953,Z 307.402,A -85,B 0,C 180,E1 -11329.416,E2 -11329.416} C_VEL
LIN {X 0,Y 552.389,Z 326.961,A -85,B 0,C 180,E1 -11331.982,E2 -11331.982} C_VEL
LIN {X 0,Y 551.777,Z 343.783,A -85,B 0,C 180,E1 -11334.171,E2 -11334.171} C_VEL
LIN {X 0,Y 555.191,Z 361.344,A -85,B 0,C 180,E1 -11334.617,E2 -11334.617} C_VEL
LIN {X 0,Y 555.624,Z 366.086,A -85,B 0,C 180,E1 -11334.715,E2 -11334.715} C_VEL
LIN {X 0,Y 553.484,Z 482.75,A -85,B 0,C 180,E1 -11336.554,E2 -11336.554} C_VEL
LIN {X 0,Y 553.086,Z 496.867,A -85,B 0,C 180,E1 -11336.915,E2 -11336.915} C_VEL
LIN {X 0,Y 552.515,Z 510.572,A -85,B 0,C 180,E1 -11337.411,E2 -11337.411} C_VEL
LIN {X 0,Y 551.962,Z 522.992,A -85,B 0,C 180,E1 -11338,E2 -11338} C_VEL
LIN {X 0,Y 551.294,Z 535.243,A -85,B 0,C 180,E1 -11338.726,E2 -11338.726} C_VEL
LIN {X 0,Y 550.698,Z 547.611,A -85,B 0,C 180,E1 -11339.636,E2 -11339.636} C_VEL
LIN {X 0,Y 550.129,Z 557.86,A -85,B 0,C 180,E1 -11340.547,E2 -11340.547} C_VEL
LIN {X 0,Y 549.421,Z 568.133,A -85,B 0,C 180,E1 -11341.644,E2 -11341.644} C_VEL
LIN {X 0,Y 548.997,Z 576.604,A -85,B 0,C 180,E1 -11342.742,E2 -11342.742} C_VEL
LIN {X 0,Y 548.449,Z 584.763,A -85,B 0,C 180,E1 -11344.028,E2 -11344.028} C_VEL
LIN {X 0,Y 548.334,Z 590.432,A -85,B 0,C 180,E1 -11345.13,E2 -11345.13} C_VEL
LIN {X 0,Y 548.129,Z 595.088,A -85,B 0,C 180,E1 -11346.236,E2 -11346.236} C_VEL
LIN {X 0,Y 547.87,Z 599.906,A -85,B 0,C 180,E1 -11347.715,E2 -11347.715} C_VEL
LIN {X 0,Y 547.814,Z 602.453,A -85,B 0,C 180,E1 -11348.826,E2 -11348.826} C_VEL
LIN {X 0,Y 547.78,Z 604.615,A -85,B 0,C 180,E1 -11350.313,E2 -11350.313} C_VEL
LIN {X 0,Y 547.644,Z 605.357,A -85,B 0,C 180,E1 -11351.809,E2 -11351.809} C_VEL
LIN {X 0,Y 547.754,Z 604.616,A -85,B 0,C 180,E1 -11353.307,E2 -11353.307} C_VEL
LIN {X 0,Y 547.709,Z 602.386,A -85,B 0,C 180,E1 -11354.819,E2 -11354.819} C_VEL
LIN {X 0,Y 547.858,Z 598.618,A -85,B 0,C 180,E1 -11356.336,E2 -11356.336} C_VEL
LIN {X 0,Y 547.959,Z 594.673,A -85,B 0,C 180,E1 -11357.481,E2 -11357.481} C_VEL
LIN {X 0,Y 548.13,Z 589.688,A -85,B 0,C 180,E1 -11358.631,E2 -11358.631} C_VEL
LIN {X 0,Y 548.358,Z 583.524,A -85,B 0,C 180,E1 -11359.785,E2 -11359.785} C_VEL
LIN {X 0,Y 548.68,Z 575.993,A -85,B 0,C 180,E1 -11360.944,E2 -11360.944} C_VEL
LIN {X 0,Y 549.054,Z 566.801,A -85,B 0,C 180,E1 -11362.107,E2 -11362.107} C_VEL
LIN {X 0,Y 549.55,Z 556.593,A -85,B 0,C 180,E1 -11363.174,E2 -11363.174} C_VEL
LIN {X 0,Y 550.049,Z 545.321,A -85,B 0,C 180,E1 -11364.147,E2 -11364.147} C_VEL
LIN {X 0,Y 550.642,Z 533.11,A -85,B 0,C 180,E1 -11365.01,E2 -11365.01} C_VEL
LIN {X 0,Y 551.091,Z 520.989,A -85,B 0,C 180,E1 -11365.705,E2 -11365.705} C_VEL
LIN {X 0,Y 551.568,Z 508.13,A -85,B 0,C 180,E1 -11366.288,E2 -11366.288} C_VEL
LIN {X 0,Y 552.003,Z 493.895,A -85,B 0,C 180,E1 -11366.773,E2 -11366.773} C_VEL
LIN {X 0,Y 552.339,Z 479.454,A -85,B 0,C 180,E1 -11367.112,E2 -11367.112} C_VEL
LIN {X 0,Y 553.816,Z 363.11,A -85,B 0,C 180,E1 -11368.836,E2 -11368.836} C_VEL
LIN {X 0,Y 550.658,Z 342.536,A -85,B 0,C 180,E1 -11369.245,E2 -11369.245} C_VEL
LIN {X 0,Y 551.356,Z 321.277,A -85,B 0,C 180,E1 -11372.072,E2 -11372.072} C_VEL
LIN {X 0,Y 551.944,Z 303.635,A -85,B 0,C 180,E1 -11374.422,E2 -11374.422} C_VEL
LIN {X 0,Y 549.529,Z 290.1,A -85,B 0,C 180,E1 -11376.327,E2 -11376.327} C_VEL
LIN {X 0,Y 549.24,Z 288.63,A -85,B 0,C 180,E1 -11376.561,E2 -11376.561} C_VEL
LIN {X 0,Y 549.148,Z 288.638,A -85,B 0,C 180,E1 -11379.625,E2 -11379.625} C_VEL
LIN {X 0,Y 549.157,Z 288.638,A -85,B 0,C 180,E1 -11382.533,E2 -11382.533} C_VEL
LIN {X 0,Y 549.206,Z 288.629,A -85,B 0,C 180,E1 -11385.454,E2 -11385.454} C_VEL
LIN {X 0,Y 549.155,Z 288.637,A -85,B 0,C 180,E1 -11388.811,E2 -11388.811} C_VEL
LIN {X 0,Y 549.134,Z 288.639,A -85,B 0,C 180,E1 -11391.315,E2 -11391.315} C_VEL
LIN {X 0,Y 549.157,Z 288.638,A -85,B 0,C 180,E1 -11394.074,E2 -11394.074} C_VEL
LIN {X 0,Y 549.131,Z 288.641,A -85,B 0,C 180,E1 -11396.735,E2 -11396.735} C_VEL
LIN {X 0,Y 549.168,Z 288.635,A -85,B 0,C 180,E1 -11399.322,E2 -11399.322} C_VEL
LIN {X 0,Y 549.19,Z 288.633,A -85,B 0,C 180,E1 -11401.841,E2 -11401.841} C_VEL
LIN {X 0,Y 549.177,Z 288.634,A -85,B 0,C 180,E1 -11404.899,E2 -11404.899} C_VEL
LIN {X 0,Y 549.201,Z 288.632,A -85,B 0,C 180,E1 -11407.503,E2 -11407.503} C_VEL
LIN {X 0,Y 549.2,Z 288.632,A -85,B 0,C 180,E1 -11409.856,E2 -11409.856} C_VEL
LIN {X 0,Y 549.192,Z 288.632,A -85,B 0,C 180,E1 -11411.54,E2 -11411.54} C_VEL
LIN {X 0,Y 548.523,Z 288.72,A -85,B 0,C 180,E1 -11412.153,E2 -11412.153} C_VEL
LIN {X 0,Y 545.679,Z 289.071,A -85,B 0,C 180,E1 -11413.147,E2 -11413.147} C_VEL
LIN {X 0,Y 543.291,Z 289.37,A -85,B 0,C 180,E1 -11413.947,E2 -11413.947} C_VEL
LIN {X 0,Y 542.282,Z 289.492,A -85,B 0,C 180,E1 -11414.565,E2 -11414.565} C_VEL
LIN {X 0,Y 542.209,Z 289.5,A -85,B 0,C 180,E1 -11414.774,E2 -11414.774} C_VEL
LIN {X 0,Y 542.191,Z 289.503,A -85,B 0,C 180,E1 -11417.312,E2 -11417.312} C_VEL
LIN {X 0,Y 542.264,Z 289.495,A -85,B 0,C 180,E1 -11419.58,E2 -11419.58} C_VEL
LIN {X 0,Y 542.319,Z 289.53,A -85,B 0,C 180,E1 -11422.484,E2 -11422.484} C_VEL
LIN {X 0,Y 543.589,Z 297.861,A -85,B 0,C 180,E1 -11424.081,E2 -11424.081} C_VEL
LIN {X 0,Y 543.47,Z 301.286,A -85,B 0,C 180,E1 -11424.706,E2 -11424.706} C_VEL
LIN {X 0,Y 547.295,Z 320.027,A -85,B 0,C 180,E1 -11425.065,E2 -11425.065} C_VEL
LIN {X 0,Y 546.087,Z 436.06,A -85,B 0,C 180,E1 -11426.597,E2 -11426.597} C_VEL
LIN {X 0,Y 545.782,Z 450.798,A -85,B 0,C 180,E1 -11426.941,E2 -11426.941} C_VEL
LIN {X 0,Y 545.4,Z 464.719,A -85,B 0,C 180,E1 -11427.422,E2 -11427.422} C_VEL
LIN {X 0,Y 544.982,Z 476.773,A -85,B 0,C 180,E1 -11427.973,E2 -11427.973} C_VEL
LIN {X 0,Y 544.55,Z 489.434,A -85,B 0,C 180,E1 -11428.708,E2 -11428.708} C_VEL
LIN {X 0,Y 543.78,Z 501.053,A -85,B 0,C 180,E1 -11429.537,E2 -11429.537} C_VEL
LIN {X 0,Y 543.297,Z 512.578,A -85,B 0,C 180,E1 -11430.552,E2 -11430.552} C_VEL
LIN {X 0,Y 542.627,Z 522.949,A -85,B 0,C 180,E1 -11431.662,E2 -11431.662} C_VEL
LIN {X 0,Y 542.187,Z 531.495,A -85,B 0,C 180,E1 -11432.775,E2 -11432.775} C_VEL
LIN {X 0,Y 541.657,Z 539.725,A -85,B 0,C 180,E1 -11434.077,E2 -11434.077} C_VEL
LIN {X 0,Y 541.534,Z 545.436,A -85,B 0,C 180,E1 -11435.193,E2 -11435.193} C_VEL
LIN {X 0,Y 541.272,Z 550.169,A -85,B 0,C 180,E1 -11436.313,E2 -11436.313} C_VEL
LIN {X 0,Y 541.019,Z 555.074,A -85,B 0,C 180,E1 -11437.811,E2 -11437.811} C_VEL
LIN {X 0,Y 540.924,Z 557.763,A -85,B 0,C 180,E1 -11438.937,E2 -11438.937} C_VEL
LIN {X 0,Y 540.881,Z 560.116,A -85,B 0,C 180,E1 -11440.444,E2 -11440.444} C_VEL
LIN {X 0,Y 540.83,Z 561.121,A -85,B 0,C 180,E1 -11441.957,E2 -11441.957} C_VEL
LIN {X 0,Y 540.923,Z 560.772,A -85,B 0,C 180,E1 -11443.477,E2 -11443.477} C_VEL
LIN {X 0,Y 540.968,Z 559.058,A -85,B 0,C 180,E1 -11445.006,E2 -11445.006} C_VEL
LIN {X 0,Y 541.206,Z 555.912,A -85,B 0,C 180,E1 -11446.541,E2 -11446.541} C_VEL
LIN {X 0,Y 541.396,Z 552.493,A -85,B 0,C 180,E1 -11447.698,E2 -11447.698} C_VEL
LIN {X 0,Y 541.833,Z 547.122,A -85,B 0,C 180,E1 -11449.1,E2 -11449.1} C_VEL
LIN {X 0,Y 542.274,Z 540.726,A -85,B 0,C 180,E1 -11450.409,E2 -11450.409} C_VEL
LIN {X 0,Y 542.818,Z 532.849,A -85,B 0,C 180,E1 -11451.708,E2 -11451.708} C_VEL
LIN {X 0,Y 543.572,Z 523.625,A -85,B 0,C 180,E1 -11452.94,E2 -11452.94} C_VEL
LIN {X 0,Y 544.287,Z 513.223,A -85,B 0,C 180,E1 -11454.075,E2 -11454.075} C_VEL
LIN {X 0,Y 545.086,Z 501.864,A -85,B 0,C 180,E1 -11455.088,E2 -11455.088} C_VEL
LIN {X 0,Y 545.806,Z 489.947,A -85,B 0,C 180,E1 -11455.957,E2 -11455.957} C_VEL
LIN {X 0,Y 546.418,Z 478.107,A -85,B 0,C 180,E1 -11456.655,E2 -11456.655} C_VEL
LIN {X 0,Y 547.015,Z 464.348,A -85,B 0,C 180,E1 -11457.293,E2 -11457.293} C_VEL
LIN {X 0,Y 547.51,Z 450.421,A -85,B 0,C 180,E1 -11457.769,E2 -11457.769} C_VEL
LIN {X 0,Y 547.771,Z 436.329,A -85,B 0,C 180,E1 -11458.096,E2 -11458.096} C_VEL
LIN {X 0,Y 549.077,Z 320.46,A -85,B 0,C 180,E1 -11459.651,E2 -11459.651} C_VEL
LIN {X 0,Y 544.828,Z 303.216,A -85,B 0,C 180,E1 -11460.061,E2 -11460.061} C_VEL
LIN {X 0,Y 544.461,Z 301.772,A -85,B 0,C 180,E1 -11460.112,E2 -11460.112} C_VEL
LIN {X 0,Y 542.118,Z 289.663,A -85,B 0,C 180,E1 -11462.587,E2 -11462.587} C_VEL
LIN {X 0,Y 542.1,Z 289.517,A -85,B 0,C 180,E1 -11465.549,E2 -11465.549} C_VEL
LIN {X 0,Y 542.074,Z 289.517,A -85,B 0,C 180,E1 -11468.33,E2 -11468.33} C_VEL
LIN {X 0,Y 542.115,Z 289.51,A -85,B 0,C 180,E1 -11471.462,E2 -11471.462} C_VEL
LIN {X 0,Y 542.133,Z 289.5,A -85,B 0,C 180,E1 -11474.716,E2 -11474.716} C_VEL
LIN {X 0,Y 542.088,Z 289.517,A -85,B 0,C 180,E1 -11477.431,E2 -11477.431} C_VEL
LIN {X 0,Y 542.111,Z 289.517,A -85,B 0,C 180,E1 -11479.757,E2 -11479.757} C_VEL
LIN {X 0,Y 542.118,Z 289.508,A -85,B 0,C 180,E1 -11482.608,E2 -11482.608} C_VEL
LIN {X 0,Y 542.112,Z 289.5,A -85,B 0,C 180,E1 -11485.354,E2 -11485.354} C_VEL
LIN {X 0,Y 542.1,Z 289.51,A -85,B 0,C 180,E1 -11488.511,E2 -11488.511} C_VEL
LIN {X 0,Y 542.128,Z 289.515,A -85,B 0,C 180,E1 -11491.442,E2 -11491.442} C_VEL
LIN {X 0,Y 542.087,Z 289.519,A -85,B 0,C 180,E1 -11493.939,E2 -11493.939} C_VEL
LIN {X 0,Y 542.117,Z 289.504,A -85,B 0,C 180,E1 -11496.536,E2 -11496.536} C_VEL
LIN {X 0,Y 542.138,Z 289.512,A -85,B 0,C 180,E1 -11499.584,E2 -11499.584} C_VEL
LIN {X 0,Y 542.124,Z 289.511,A -85,B 0,C 180,E1 -11501.935,E2 -11501.935} C_VEL
LIN {X 0,Y 542.187,Z 289.504,A -85,B 0,C 180,E1 -11505.026,E2 -11505.026} C_VEL
LIN {X 0,Y 542.178,Z 289.503,A -85,B 0,C 180,E1 -11508.071,E2 -11508.071} C_VEL
LIN {X 0,Y 542.164,Z 289.499,A -85,B 0,C 180,E1 -11510.331,E2 -11510.331} C_VEL
LIN {X 0,Y 542.263,Z 289.49,A -85,B 0,C 180,E1 -11512.578,E2 -11512.578} C_VEL
LIN {X 0,Y 542.309,Z 289.489,A -85,B 0,C 180,E1 -11514.813,E2 -11514.813} C_VEL
LIN {X 0,Y 542.131,Z 289.505,A -85,B 0,C 180,E1 -11517.038,E2 -11517.038} C_VEL
LIN {X 0,Y 542.459,Z 289.474,A -85,B 0,C 180,E1 -11519.26,E2 -11519.26} C_VEL
LIN {X 0,Y 542.322,Z 289.478,A -85,B 0,C 180,E1 -11521.48,E2 -11521.48} C_VEL
LIN {X 0,Y 542.328,Z 289.485,A -85,B 0,C 180,E1 -11524.445,E2 -11524.445} C_VEL
LIN {X 0,Y 542.258,Z 289.493,A -85,B 0,C 180,E1 -11526.676,E2 -11526.676} C_VEL
LIN {X 0,Y 542.197,Z 289.499,A -85,B 0,C 180,E1 -11529.668,E2 -11529.668} C_VEL
LIN {X 0,Y 542.199,Z 289.493,A -85,B 0,C 180,E1 -11531.929,E2 -11531.929} C_VEL
LIN {X 0,Y 542.199,Z 289.504,A -85,B 0,C 180,E1 -11534.973,E2 -11534.973} C_VEL
LIN {X 0,Y 542.162,Z 289.498,A -85,B 0,C 180,E1 -11537.286,E2 -11537.286} C_VEL
LIN {X 0,Y 542.126,Z 289.508,A -85,B 0,C 180,E1 -11539.629,E2 -11539.629} C_VEL
LIN {X 0,Y 542.114,Z 289.505,A -85,B 0,C 180,E1 -11542.006,E2 -11542.006} C_VEL
LIN {X 0,Y 542.119,Z 289.515,A -85,B 0,C 180,E1 -11544.422,E2 -11544.422} C_VEL
LIN {X 0,Y 542.133,Z 289.507,A -85,B 0,C 180,E1 -11547.718,E2 -11547.718} C_VEL
LIN {X 0,Y 542.131,Z 289.511,A -85,B 0,C 180,E1 -11550.258,E2 -11550.258} C_VEL
LIN {X 0,Y 542.14,Z 289.509,A -85,B 0,C 180,E1 -11552.886,E2 -11552.886} C_VEL
LIN {X 0,Y 542.173,Z 289.485,A -85,B 0,C 180,E1 -11555.547,E2 -11555.547} C_VEL
LIN {X 0,Y 542.154,Z 289.51,A -85,B 0,C 180,E1 -11558.327,E2 -11558.327} C_VEL
LIN {X 0,Y 542.131,Z 289.509,A -85,B 0,C 180,E1 -11561.468,E2 -11561.468} C_VEL
LIN {X 0,Y 542.137,Z 289.515,A -85,B 0,C 180,E1 -11564.242,E2 -11564.242} C_VEL
LIN {X 0,Y 542.142,Z 289.508,A -85,B 0,C 180,E1 -11566.787,E2 -11566.787} C_VEL
LIN {X 0,Y 542.147,Z 289.51,A -85,B 0,C 180,E1 -11569.763,E2 -11569.763} C_VEL
LIN {X 0,Y 542.177,Z 289.505,A -85,B 0,C 180,E1 -11572.616,E2 -11572.616} C_VEL
LIN {X 0,Y 542.148,Z 289.514,A -85,B 0,C 180,E1 -11575.359,E2 -11575.359} C_VEL
LIN {X 0,Y 542.116,Z 289.521,A -85,B 0,C 180,E1 -11578.513,E2 -11578.513} C_VEL
LIN {X 0,Y 542.135,Z 289.516,A -85,B 0,C 180,E1 -11581.47,E2 -11581.47} C_VEL
LIN {X 0,Y 542.185,Z 289.733,A -85,B 0,C 180,E1 -11581.819,E2 -11581.819} C_VEL
LIN {X 0,Y 545.702,Z 305.47,A -85,B 0,C 180,E1 -11584.331,E2 -11584.331} C_VEL
LIN {X 0,Y 546.625,Z 310.796,A -85,B 0,C 180,E1 -11585.149,E2 -11585.149} C_VEL
LIN {X 0,Y 545.374,Z 330.183,A -85,B 0,C 180,E1 -11587.863,E2 -11587.863} C_VEL
LIN {X 0,Y 544.061,Z 351.801,A -85,B 0,C 180,E1 -11590.837,E2 -11590.837} C_VEL
LIN {X 0,Y 543.631,Z 359.728,A -85,B 0,C 180,E1 -11591.917,E2 -11591.917} C_VEL
LIN {X 0,Y 547.542,Z 384.67,A -85,B 0,C 180,E1 -11592.411,E2 -11592.411} C_VEL
LIN {X 0,Y 548.467,Z 393.353,A -85,B 0,C 180,E1 -11592.565,E2 -11592.565} C_VEL
LIN {X 0,Y 547.243,Z 497.913,A -85,B 0,C 180,E1 -11593.968,E2 -11593.968} C_VEL
LIN {X 0,Y 546.734,Z 512.367,A -85,B 0,C 180,E1 -11594.307,E2 -11594.307} C_VEL
LIN {X 0,Y 546.065,Z 525.61,A -85,B 0,C 180,E1 -11594.757,E2 -11594.757} C_VEL
LIN {X 0,Y 545.358,Z 537.89,A -85,B 0,C 180,E1 -11595.308,E2 -11595.308} C_VEL
LIN {X 0,Y 544.569,Z 550.784,A -85,B 0,C 180,E1 -11596.047,E2 -11596.047} C_VEL
LIN {X 0,Y 543.685,Z 562.509,A -85,B 0,C 180,E1 -11596.878,E2 -11596.878} C_VEL
LIN {X 0,Y 542.874,Z 574.242,A -85,B 0,C 180,E1 -11597.899,E2 -11597.899} C_VEL
LIN {X 0,Y 542.315,Z 584.532,A -85,B 0,C 180,E1 -11598.993,E2 -11598.993} C_VEL
LIN {X 0,Y 541.688,Z 593.468,A -85,B 0,C 180,E1 -11600.137,E2 -11600.137} C_VEL
LIN {X 0,Y 541.21,Z 601.856,A -85,B 0,C 180,E1 -11601.443,E2 -11601.443} C_VEL
LIN {X 0,Y 540.877,Z 611.539,A -85,B 0,C 180,E1 -11603.309,E2 -11603.309} C_VEL
LIN {X 0,Y 540.803,Z 616.479,A -85,B 0,C 180,E1 -11604.427,E2 -11604.427} C_VEL
LIN {X 0,Y 540.732,Z 621.463,A -85,B 0,C 180,E1 -11605.892,E2 -11605.892} C_VEL
LIN {X 0,Y 540.744,Z 624.271,A -85,B 0,C 180,E1 -11607.032,E2 -11607.032} C_VEL
LIN {X 0,Y 540.714,Z 626.609,A -85,B 0,C 180,E1 -11608.517,E2 -11608.517} C_VEL
LIN {X 0,Y 540.715,Z 627.516,A -85,B 0,C 180,E1 -11610.002,E2 -11610.002} C_VEL
LIN {X 0,Y 540.713,Z 627.003,A -85,B 0,C 180,E1 -11611.486,E2 -11611.486} C_VEL
LIN {X 0,Y 540.728,Z 625.069,A -85,B 0,C 180,E1 -11612.972,E2 -11612.972} C_VEL
LIN {X 0,Y 540.74,Z 621.637,A -85,B 0,C 180,E1 -11614.459,E2 -11614.459} C_VEL
LIN {X 0,Y 540.822,Z 618.047,A -85,B 0,C 180,E1 -11615.576,E2 -11615.576} C_VEL
LIN {X 0,Y 540.937,Z 613.496,A -85,B 0,C 180,E1 -11616.694,E2 -11616.694} C_VEL
LIN {X 0,Y 541.154,Z 606.9,A -85,B 0,C 180,E1 -11618,E2 -11618} C_VEL
LIN {X 0,Y 541.524,Z 599.948,A -85,B 0,C 180,E1 -11619.119,E2 -11619.119} C_VEL
LIN {X 0,Y 541.861,Z 591.593,A -85,B 0,C 180,E1 -11620.24,E2 -11620.24} C_VEL
LIN {X 0,Y 542.475,Z 581.514,A -85,B 0,C 180,E1 -11621.358,E2 -11621.358} C_VEL
LIN {X 0,Y 543.068,Z 570.322,A -85,B 0,C 180,E1 -11622.384,E2 -11622.384} C_VEL
LIN {X 0,Y 543.766,Z 557.788,A -85,B 0,C 180,E1 -11623.314,E2 -11623.314} C_VEL
LIN {X 0,Y 544.413,Z 545.406,A -85,B 0,C 180,E1 -11624.056,E2 -11624.056} C_VEL
LIN {X 0,Y 545.055,Z 531.7,A -85,B 0,C 180,E1 -11624.704,E2 -11624.704} C_VEL
LIN {X 0,Y 545.603,Z 518.136,A -85,B 0,C 180,E1 -11625.189,E2 -11625.189} C_VEL
LIN {X 0,Y 546.092,Z 503.333,A -85,B 0,C 180,E1 -11625.556,E2 -11625.556} C_VEL
LIN {X 0,Y 548.164,Z 392.054,A -85,B 0,C 180,E1 -11627.348,E2 -11627.348} C_VEL
LIN {X 0,Y 545.333,Z 367.728,A -85,B 0,C 180,E1 -11627.9,E2 -11627.9} C_VEL
LIN {X 0,Y 543.226,Z 353.843,A -85,B 0,C 180,E1 -11628.271,E2 -11628.271} C_VEL
LIN {X 0,Y 544.376,Z 329.541,A -85,B 0,C 180,E1 -11631.514,E2 -11631.514} C_VEL
LIN {X 0,Y 545.593,Z 307.744,A -85,B 0,C 180,E1 -11634.46,E2 -11634.46} C_VEL
LIN {X 0,Y 543.395,Z 295.79,A -85,B 0,C 180,E1 -11636.2,E2 -11636.2} C_VEL
LIN {X 0,Y 542.194,Z 289.506,A -85,B 0,C 180,E1 -11637.156,E2 -11637.156} C_VEL
LIN {X 0,Y 542.128,Z 289.511,A -85,B 0,C 180,E1 -11640.259,E2 -11640.259} C_VEL
LIN {X 0,Y 542.093,Z 289.513,A -85,B 0,C 180,E1 -11642.873,E2 -11642.873} C_VEL
LIN {X 0,Y 542.118,Z 289.517,A -85,B 0,C 180,E1 -11645.552,E2 -11645.552} C_VEL
LIN {X 0,Y 542.088,Z 289.516,A -85,B 0,C 180,E1 -11648.334,E2 -11648.334} C_VEL
LIN {X 0,Y 542.107,Z 289.516,A -85,B 0,C 180,E1 -11651.222,E2 -11651.222} C_VEL
LIN {X 0,Y 542.119,Z 289.511,A -85,B 0,C 180,E1 -11654.245,E2 -11654.245} C_VEL
LIN {X 0,Y 542.081,Z 289.519,A -85,B 0,C 180,E1 -11656.777,E2 -11656.777} C_VEL
LIN {X 0,Y 542.124,Z 289.51,A -85,B 0,C 180,E1 -11659.758,E2 -11659.758} C_VEL
LIN {X 0,Y 542.127,Z 289.516,A -85,B 0,C 180,E1 -11662.609,E2 -11662.609} C_VEL
LIN {X 0,Y 542.136,Z 289.51,A -85,B 0,C 180,E1 -11665.355,E2 -11665.355} C_VEL
LIN {X 0,Y 542.117,Z 289.517,A -85,B 0,C 180,E1 -11668.515,E2 -11668.515} C_VEL
LIN {X 0,Y 542.145,Z 289.508,A -85,B 0,C 180,E1 -11671.47,E2 -11671.47} C_VEL
LIN {X 0,Y 542.117,Z 289.516,A -85,B 0,C 180,E1 -11673.941,E2 -11673.941} C_VEL
LIN {X 0,Y 542.148,Z 289.517,A -85,B 0,C 180,E1 -11676.538,E2 -11676.538} C_VEL
LIN {X 0,Y 542.169,Z 289.515,A -85,B 0,C 180,E1 -11679.585,E2 -11679.585} C_VEL
LIN {X 0,Y 542.153,Z 289.517,A -85,B 0,C 180,E1 -11681.936,E2 -11681.936} C_VEL
LIN {X 0,Y 542.188,Z 289.507,A -85,B 0,C 180,E1 -11685.026,E2 -11685.026} C_VEL
LIN {X 0,Y 542.232,Z 289.51,A -85,B 0,C 180,E1 -11686.412,E2 -11686.412} C_VEL
LIN {X 0,Y 545.48,Z 303.693,A -85,B 0,C 180,E1 -11688.52,E2 -11688.52} C_VEL
LIN {X 0,Y 546.187,Z 309.059,A -85,B 0,C 180,E1 -11689.283,E2 -11689.283} C_VEL
LIN {X 0,Y 545.573,Z 328.75,A -85,B 0,C 180,E1 -11691.881,E2 -11691.881} C_VEL
LIN {X 0,Y 544.943,Z 343.791,A -85,B 0,C 180,E1 -11693.866,E2 -11693.866} C_VEL
LIN {X 0,Y 548.503,Z 361.73,A -85,B 0,C 180,E1 -11694.342,E2 -11694.342} C_VEL
LIN {X 0,Y 549.018,Z 367.201,A -85,B 0,C 180,E1 -11694.459,E2 -11694.459} C_VEL
LIN {X 0,Y 546.763,Z 483.136,A -85,B 0,C 180,E1 -11696.327,E2 -11696.327} C_VEL
LIN {X 0,Y 546.329,Z 497.125,A -85,B 0,C 180,E1 -11696.693,E2 -11696.693} C_VEL
LIN {X 0,Y 545.74,Z 510.758,A -85,B 0,C 180,E1 -11697.195,E2 -11697.195} C_VEL
LIN {X 0,Y 545.134,Z 523.169,A -85,B 0,C 180,E1 -11697.791,E2 -11697.791} C_VEL
LIN {X 0,Y 544.454,Z 535.417,A -85,B 0,C 180,E1 -11698.526,E2 -11698.526} C_VEL
LIN {X 0,Y 543.806,Z 547.794,A -85,B 0,C 180,E1 -11699.446,E2 -11699.446} C_VEL
LIN {X 0,Y 543.228,Z 558.021,A -85,B 0,C 180,E1 -11700.369,E2 -11700.369} C_VEL
LIN {X 0,Y 542.451,Z 568.294,A -85,B 0,C 180,E1 -11701.48,E2 -11701.48} C_VEL
LIN {X 0,Y 541.993,Z 576.767,A -85,B 0,C 180,E1 -11702.592,E2 -11702.592} C_VEL
LIN {X 0,Y 541.404,Z 584.936,A -85,B 0,C 180,E1 -11703.895,E2 -11703.895} C_VEL
LIN {X 0,Y 541.246,Z 591.443,A -85,B 0,C 180,E1 -11705.197,E2 -11705.197} C_VEL
LIN {X 0,Y 540.962,Z 597.236,A -85,B 0,C 180,E1 -11706.692,E2 -11706.692} C_VEL
LIN {X 0,Y 540.716,Z 601.446,A -85,B 0,C 180,E1 -11708.192,E2 -11708.192} C_VEL
LIN {X 0,Y 540.716,Z 604.154,A -85,B 0,C 180,E1 -11709.695,E2 -11709.695} C_VEL
LIN {X 0,Y 540.606,Z 605.4,A -85,B 0,C 180,E1 -11711.207,E2 -11711.207} C_VEL
LIN {X 0,Y 540.604,Z 605.191,A -85,B 0,C 180,E1 -11712.725,E2 -11712.725} C_VEL
LIN {X 0,Y 540.661,Z 604.332,A -85,B 0,C 180,E1 -11713.672,E2 -11713.672} C_VEL
LIN {X 0,Y 540.636,Z 602.126,A -85,B 0,C 180,E1 -11715.018,E2 -11715.018} C_VEL
LIN {X 0,Y 540.796,Z 598.158,A -85,B 0,C 180,E1 -11716.556,E2 -11716.556} C_VEL
LIN {X 0,Y 540.899,Z 594.006,A -85,B 0,C 180,E1 -11717.717,E2 -11717.717} C_VEL
LIN {X 0,Y 541.172,Z 587.647,A -85,B 0,C 180,E1 -11719.115,E2 -11719.115} C_VEL
LIN {X 0,Y 541.412,Z 579.95,A -85,B 0,C 180,E1 -11720.445,E2 -11720.445} C_VEL
LIN {X 0,Y 541.845,Z 571.14,A -85,B 0,C 180,E1 -11721.677,E2 -11721.677} C_VEL
LIN {X 0,Y 542.294,Z 561.409,A -85,B 0,C 180,E1 -11722.798,E2 -11722.798} C_VEL
LIN {X 0,Y 542.82,Z 550.431,A -85,B 0,C 180,E1 -11723.843,E2 -11723.843} C_VEL
LIN {X 0,Y 543.366,Z 538.58,A -85,B 0,C 180,E1 -11724.768,E2 -11724.768} C_VEL
LIN {X 0,Y 543.914,Z 525.599,A -85,B 0,C 180,E1 -11725.585,E2 -11725.585} C_VEL
LIN {X 0,Y 544.425,Z 512.298,A -85,B 0,C 180,E1 -11726.248,E2 -11726.248} C_VEL
LIN {X 0,Y 544.901,Z 498.069,A -85,B 0,C 180,E1 -11726.789,E2 -11726.789} C_VEL
LIN {X 0,Y 545.376,Z 483.627,A -85,B 0,C 180,E1 -11727.177,E2 -11727.177} C_VEL
LIN {X 0,Y 545.644,Z 459.277,A -85,B 0,C 180,E1 -11727.57,E2 -11727.57} C_VEL
LIN {X 0,Y 546.916,Z 363.872,A -85,B 0,C 180,E1 -11729.004,E2 -11729.004} C_VEL
LIN {X 0,Y 543.702,Z 342.632,A -85,B 0,C 180,E1 -11729.43,E2 -11729.43} C_VEL
LIN {X 0,Y 544.422,Z 321.778,A -85,B 0,C 180,E1 -11732.228,E2 -11732.228} C_VEL
LIN {X 0,Y 544.895,Z 303.796,A -85,B 0,C 180,E1 -11734.642,E2 -11734.642} C_VEL
LIN {X 0,Y 542.204,Z 289.506,A -85,B 0,C 180,E1 -11736.71,E2 -11736.71} C_VEL
LIN {X 0,Y 542.124,Z 289.517,A -85,B 0,C 180,E1 -11740.242,E2 -11740.242} C_VEL
LIN {X 0,Y 542.13,Z 289.51,A -85,B 0,C 180,E1 -11743.218,E2 -11743.218} C_VEL
LIN {X 0,Y 542.151,Z 289.509,A -85,B 0,C 180,E1 -11745.758,E2 -11745.758} C_VEL
LIN {X 0,Y 542.108,Z 289.515,A -85,B 0,C 180,E1 -11748.778,E2 -11748.778} C_VEL
LIN {X 0,Y 542.081,Z 289.519,A -85,B 0,C 180,E1 -11751.666,E2 -11751.666} C_VEL
LIN {X 0,Y 542.119,Z 289.514,A -85,B 0,C 180,E1 -11754.488,E2 -11754.488} C_VEL
LIN {X 0,Y 542.104,Z 289.514,A -85,B 0,C 180,E1 -11757.133,E2 -11757.133} C_VEL
LIN {X 0,Y 542.133,Z 289.513,A -85,B 0,C 180,E1 -11759.957,E2 -11759.957} C_VEL
LIN {X 0,Y 542.138,Z 289.513,A -85,B 0,C 180,E1 -11762.28,E2 -11762.28} C_VEL
LIN {X 0,Y 542.143,Z 289.511,A -85,B 0,C 180,E1 -11765.578,E2 -11765.578} C_VEL
LIN {X 0,Y 542.178,Z 289.508,A -85,B 0,C 180,E1 -11768.462,E2 -11768.462} C_VEL
LIN {X 0,Y 542.15,Z 289.508,A -85,B 0,C 180,E1 -11771.54,E2 -11771.54} C_VEL
LIN {X 0,Y 542.211,Z 289.504,A -85,B 0,C 180,E1 -11774.258,E2 -11774.258} C_VEL
LIN {X 0,Y 542.209,Z 289.5,A -85,B 0,C 180,E1 -11774.774,E2 -11774.774} C_VEL
LIN {X 0,Y 541.561,Z 289.582,A -85,B 0,C 180,E1 -11775.394,E2 -11775.394} C_VEL
LIN {X 0,Y 538.696,Z 289.945,A -85,B 0,C 180,E1 -11776.4,E2 -11776.4} C_VEL
LIN {X 0,Y 536.266,Z 290.25,A -85,B 0,C 180,E1 -11777.209,E2 -11777.209} C_VEL
LIN {X 0,Y 535.23,Z 290.375,A -85,B 0,C 180,E1 -11777.835,E2 -11777.835} C_VEL
LIN {X 0,Y 535.151,Z 290.383,A -85,B 0,C 180,E1 -11778.047,E2 -11778.047} C_VEL
LIN {X 0,Y 535.167,Z 290.383,A -85,B 0,C 180,E1 -11780.202,E2 -11780.202} C_VEL
LIN {X 0,Y 535.283,Z 290.555,A -85,B 0,C 180,E1 -11782.385,E2 -11782.385} C_VEL
LIN {X 0,Y 536.594,Z 298.918,A -85,B 0,C 180,E1 -11784.004,E2 -11784.004} C_VEL
LIN {X 0,Y 536.556,Z 301.577,A -85,B 0,C 180,E1 -11784.497,E2 -11784.497} C_VEL
LIN {X 0,Y 540.438,Z 320.938,A -85,B 0,C 180,E1 -11784.886,E2 -11784.886} C_VEL
LIN {X 0,Y 539.173,Z 436.856,A -85,B 0,C 180,E1 -11786.437,E2 -11786.437} C_VEL
LIN {X 0,Y 538.856,Z 451.432,A -85,B 0,C 180,E1 -11786.785,E2 -11786.785} C_VEL
LIN {X 0,Y 538.486,Z 464.739,A -85,B 0,C 180,E1 -11787.249,E2 -11787.249} C_VEL
LIN {X 0,Y 538.022,Z 477.75,A -85,B 0,C 180,E1 -11787.853,E2 -11787.853} C_VEL
LIN {X 0,Y 537.549,Z 490.314,A -85,B 0,C 180,E1 -11788.598,E2 -11788.598} C_VEL
LIN {X 0,Y 536.779,Z 501.849,A -85,B 0,C 180,E1 -11789.437,E2 -11789.437} C_VEL
LIN {X 0,Y 536.352,Z 512.344,A -85,B 0,C 180,E1 -11790.372,E2 -11790.372} C_VEL
LIN {X 0,Y 535.635,Z 522.828,A -85,B 0,C 180,E1 -11791.497,E2 -11791.497} C_VEL
LIN {X 0,Y 535.155,Z 531.468,A -85,B 0,C 180,E1 -11792.624,E2 -11792.624} C_VEL
LIN {X 0,Y 534.692,Z 538.674,A -85,B 0,C 180,E1 -11793.754,E2 -11793.754} C_VEL
LIN {X 0,Y 534.478,Z 545.815,A -85,B 0,C 180,E1 -11795.128,E2 -11795.128} C_VEL
LIN {X 0,Y 534.197,Z 551.055,A -85,B 0,C 180,E1 -11796.397,E2 -11796.397} C_VEL
LIN {X 0,Y 533.926,Z 555.845,A -85,B 0,C 180,E1 -11797.916,E2 -11797.916} C_VEL
LIN {X 0,Y 533.855,Z 558.42,A -85,B 0,C 180,E1 -11799.057,E2 -11799.057} C_VEL
LIN {X 0,Y 533.803,Z 560.666,A -85,B 0,C 180,E1 -11800.584,E2 -11800.584} C_VEL
LIN {X 0,Y 533.739,Z 561.566,A -85,B 0,C 180,E1 -11802.119,E2 -11802.119} C_VEL
LIN {X 0,Y 533.864,Z 561.108,A -85,B 0,C 180,E1 -11803.658,E2 -11803.658} C_VEL
LIN {X 0,Y 533.923,Z 559.284,A -85,B 0,C 180,E1 -11805.209,E2 -11805.209} C_VEL
LIN {X 0,Y 534.204,Z 555.983,A -85,B 0,C 180,E1 -11806.764,E2 -11806.764} C_VEL
LIN {X 0,Y 534.519,Z 551.1,A -85,B 0,C 180,E1 -11808.328,E2 -11808.328} C_VEL
LIN {X 0,Y 534.937,Z 545.861,A -85,B 0,C 180,E1 -11809.604,E2 -11809.604} C_VEL
LIN {X 0,Y 535.387,Z 539.32,A -85,B 0,C 180,E1 -11810.884,E2 -11810.884} C_VEL
LIN {X 0,Y 535.971,Z 532.31,A -85,B 0,C 180,E1 -11812.01,E2 -11812.01} C_VEL
LIN {X 0,Y 536.72,Z 522.926,A -85,B 0,C 180,E1 -11813.25,E2 -11813.25} C_VEL
LIN {X 0,Y 537.454,Z 513.266,A -85,B 0,C 180,E1 -11814.303,E2 -11814.303} C_VEL
LIN {X 0,Y 538.293,Z 501.885,A -85,B 0,C 180,E1 -11815.324,E2 -11815.324} C_VEL
LIN {X 0,Y 539.06,Z 489.698,A -85,B 0,C 180,E1 -11816.216,E2 -11816.216} C_VEL
LIN {X 0,Y 539.789,Z 476.09,A -85,B 0,C 180,E1 -11817.009,E2 -11817.009} C_VEL
LIN {X 0,Y 540.358,Z 462.743,A -85,B 0,C 180,E1 -11817.605,E2 -11817.605} C_VEL
LIN {X 0,Y 540.785,Z 448.408,A -85,B 0,C 180,E1 -11818.074,E2 -11818.074} C_VEL
LIN {X 0,Y 541.1,Z 433.766,A -85,B 0,C 180,E1 -11818.385,E2 -11818.385} C_VEL
LIN {X 0,Y 542.401,Z 321.377,A -85,B 0,C 180,E1 -11819.907,E2 -11819.907} C_VEL
LIN {X 0,Y 538.45,Z 305.345,A -85,B 0,C 180,E1 -11820.296,E2 -11820.296} C_VEL
LIN {X 0,Y 537.391,Z 302.222,A -85,B 0,C 180,E1 -11820.393,E2 -11820.393} C_VEL
LIN {X 0,Y 535.075,Z 290.514,A -85,B 0,C 180,E1 -11822.821,E2 -11822.821} C_VEL
LIN {X 0,Y 535.062,Z 290.396,A -85,B 0,C 180,E1 -11825.744,E2 -11825.744} C_VEL
LIN {X 0,Y 535.037,Z 290.395,A -85,B 0,C 180,E1 -11828.234,E2 -11828.234} C_VEL
LIN {X 0,Y 535.042,Z 290.392,A -85,B 0,C 180,E1 -11830.884,E2 -11830.884} C_VEL
LIN {X 0,Y 535.081,Z 290.389,A -85,B 0,C 180,E1 -11833.948,E2 -11833.948} C_VEL
LIN {X 0,Y 535.068,Z 290.39,A -85,B 0,C 180,E1 -11837.142,E2 -11837.142} C_VEL
LIN {X 0,Y 535.064,Z 290.393,A -85,B 0,C 180,E1 -11840.1,E2 -11840.1} C_VEL
LIN {X 0,Y 535.083,Z 290.384,A -85,B 0,C 180,E1 -11842.984,E2 -11842.984} C_VEL
LIN {X 0,Y 535.059,Z 290.384,A -85,B 0,C 180,E1 -11845.743,E2 -11845.743} C_VEL
LIN {X 0,Y 535.057,Z 290.388,A -85,B 0,C 180,E1 -11848.423,E2 -11848.423} C_VEL
LIN {X 0,Y 535.077,Z 290.391,A -85,B 0,C 180,E1 -11851.285,E2 -11851.285} C_VEL
LIN {X 0,Y 535.061,Z 290.391,A -85,B 0,C 180,E1 -11853.571,E2 -11853.571} C_VEL
LIN {X 0,Y 535.072,Z 290.382,A -85,B 0,C 180,E1 -11856.391,E2 -11856.391} C_VEL
LIN {X 0,Y 535.11,Z 290.389,A -85,B 0,C 180,E1 -11859.303,E2 -11859.303} C_VEL
LIN {X 0,Y 535.07,Z 290.389,A -85,B 0,C 180,E1 -11861.689,E2 -11861.689} C_VEL
LIN {X 0,Y 535.113,Z 290.383,A -85,B 0,C 180,E1 -11864.045,E2 -11864.045} C_VEL
LIN {X 0,Y 535.159,Z 290.37,A -85,B 0,C 180,E1 -11866.373,E2 -11866.373} C_VEL
LIN {X 0,Y 535.203,Z 290.374,A -85,B 0,C 180,E1 -11869.442,E2 -11869.442} C_VEL
LIN {X 0,Y 535.231,Z 290.365,A -85,B 0,C 180,E1 -11872.48,E2 -11872.48} C_VEL
LIN {X 0,Y 535.26,Z 290.367,A -85,B 0,C 180,E1 -11874.744,E2 -11874.744} C_VEL
LIN {X 0,Y 535.273,Z 290.353,A -85,B 0,C 180,E1 -11876.249,E2 -11876.249} C_VEL
LIN {X 0,Y 535.408,Z 290.352,A -85,B 0,C 180,E1 -11879.25,E2 -11879.25} C_VEL
LIN {X 0,Y 535.269,Z 290.356,A -85,B 0,C 180,E1 -11881.5,E2 -11881.5} C_VEL
LIN {X 0,Y 535.295,Z 290.361,A -85,B 0,C 180,E1 -11884.503,E2 -11884.503} C_VEL
LIN {X 0,Y 535.235,Z 290.366,A -85,B 0,C 180,E1 -11886.764,E2 -11886.764} C_VEL
LIN {X 0,Y 535.172,Z 290.374,A -85,B 0,C 180,E1 -11889.796,E2 -11889.796} C_VEL
LIN {X 0,Y 535.145,Z 290.372,A -85,B 0,C 180,E1 -11892.089,E2 -11892.089} C_VEL
LIN {X 0,Y 535.185,Z 290.372,A -85,B 0,C 180,E1 -11894.429,E2 -11894.429} C_VEL
LIN {X 0,Y 535.116,Z 290.373,A -85,B 0,C 180,E1 -11897.521,E2 -11897.521} C_VEL
LIN {X 0,Y 535.111,Z 290.387,A -85,B 0,C 180,E1 -11900.697,E2 -11900.697} C_VEL
LIN {X 0,Y 535.074,Z 290.387,A -85,B 0,C 180,E1 -11903.942,E2 -11903.942} C_VEL
LIN {X 0,Y 535.062,Z 290.389,A -85,B 0,C 180,E1 -11906.429,E2 -11906.429} C_VEL
LIN {X 0,Y 535.077,Z 290.389,A -85,B 0,C 180,E1 -11908.97,E2 -11908.97} C_VEL
LIN {X 0,Y 535.076,Z 290.387,A -85,B 0,C 180,E1 -11911.697,E2 -11911.697} C_VEL
LIN {X 0,Y 535.084,Z 290.377,A -85,B 0,C 180,E1 -11914.447,E2 -11914.447} C_VEL
LIN {X 0,Y 535.146,Z 290.375,A -85,B 0,C 180,E1 -11917.025,E2 -11917.025} C_VEL
LIN {X 0,Y 535.093,Z 290.388,A -85,B 0,C 180,E1 -11919.898,E2 -11919.898} C_VEL
LIN {X 0,Y 535.077,Z 290.388,A -85,B 0,C 180,E1 -11922.899,E2 -11922.899} C_VEL
LIN {X 0,Y 535.083,Z 290.385,A -85,B 0,C 180,E1 -11925.022,E2 -11925.022} C_VEL
LIN {X 0,Y 535.115,Z 290.389,A -85,B 0,C 180,E1 -11928.124,E2 -11928.124} C_VEL
LIN {X 0,Y 535.078,Z 290.388,A -85,B 0,C 180,E1 -11931.075,E2 -11931.075} C_VEL
LIN {X 0,Y 535.126,Z 290.382,A -85,B 0,C 180,E1 -11933.915,E2 -11933.915} C_VEL
LIN {X 0,Y 535.081,Z 290.394,A -85,B 0,C 180,E1 -11936.907,E2 -11936.907} C_VEL
LIN {X 0,Y 535.09,Z 290.397,A -85,B 0,C 180,E1 -11939.764,E2 -11939.764} C_VEL
LIN {X 0,Y 535.126,Z 290.509,A -85,B 0,C 180,E1 -11941.535,E2 -11941.535} C_VEL
LIN {X 0,Y 538.348,Z 304.807,A -85,B 0,C 180,E1 -11943.865,E2 -11943.865} C_VEL
LIN {X 0,Y 539.78,Z 312.559,A -85,B 0,C 180,E1 -11945.08,E2 -11945.08} C_VEL
LIN {X 0,Y 538.39,Z 332.017,A -85,B 0,C 180,E1 -11947.836,E2 -11947.836} C_VEL
LIN {X 0,Y 537.086,Z 353.063,A -85,B 0,C 180,E1 -11950.776,E2 -11950.776} C_VEL
LIN {X 0,Y 536.739,Z 359.224,A -85,B 0,C 180,E1 -11951.627,E2 -11951.627} C_VEL
LIN {X 0,Y 540.93,Z 385.825,A -85,B 0,C 180,E1 -11952.174,E2 -11952.174} C_VEL
LIN {X 0,Y 541.768,Z 394.222,A -85,B 0,C 180,E1 -11952.323,E2 -11952.323} C_VEL
LIN {X 0,Y 540.522,Z 497.725,A -85,B 0,C 180,E1 -11953.732,E2 -11953.732} C_VEL
LIN {X 0,Y 539.972,Z 511.99,A -85,B 0,C 180,E1 -11954.07,E2 -11954.07} C_VEL
LIN {X 0,Y 539.24,Z 526.025,A -85,B 0,C 180,E1 -11954.559,E2 -11954.559} C_VEL
LIN {X 0,Y 538.427,Z 539.877,A -85,B 0,C 180,E1 -11955.211,E2 -11955.211} C_VEL
LIN {X 0,Y 537.571,Z 552.302,A -85,B 0,C 180,E1 -11955.957,E2 -11955.957} C_VEL
LIN {X 0,Y 536.679,Z 563.681,A -85,B 0,C 180,E1 -11956.799,E2 -11956.799} C_VEL
LIN {X 0,Y 535.911,Z 574.168,A -85,B 0,C 180,E1 -11957.74,E2 -11957.74} C_VEL
LIN {X 0,Y 535.258,Z 585.274,A -85,B 0,C 180,E1 -11958.95,E2 -11958.95} C_VEL
LIN {X 0,Y 534.581,Z 594.586,A -85,B 0,C 180,E1 -11960.195,E2 -11960.195} C_VEL
LIN {X 0,Y 534.106,Z 602.65,A -85,B 0,C 180,E1 -11961.518,E2 -11961.518} C_VEL
LIN {X 0,Y 533.771,Z 612.95,A -85,B 0,C 180,E1 -11963.598,E2 -11963.598} C_VEL
LIN {X 0,Y 533.729,Z 617.608,A -85,B 0,C 180,E1 -11964.731,E2 -11964.731} C_VEL
LIN {X 0,Y 533.642,Z 621.635,A -85,B 0,C 180,E1 -11965.994,E2 -11965.994} C_VEL
LIN {X 0,Y 533.643,Z 624.036,A -85,B 0,C 180,E1 -11966.992,E2 -11966.992} C_VEL
LIN {X 0,Y 533.638,Z 626.415,A -85,B 0,C 180,E1 -11968.498,E2 -11968.498} C_VEL
LIN {X 0,Y 533.632,Z 627.358,A -85,B 0,C 180,E1 -11970.002,E2 -11970.002} C_VEL
LIN {X 0,Y 533.638,Z 626.876,A -85,B 0,C 180,E1 -11971.506,E2 -11971.506} C_VEL
LIN {X 0,Y 533.629,Z 624.972,A -85,B 0,C 180,E1 -11973.011,E2 -11973.011} C_VEL
LIN {X 0,Y 533.667,Z 621.585,A -85,B 0,C 180,E1 -11974.519,E2 -11974.519} C_VEL
LIN {X 0,Y 533.746,Z 618.009,A -85,B 0,C 180,E1 -11975.65,E2 -11975.65} C_VEL
LIN {X 0,Y 533.855,Z 613.489,A -85,B 0,C 180,E1 -11976.783,E2 -11976.783} C_VEL
LIN {X 0,Y 534.103,Z 606.92,A -85,B 0,C 180,E1 -11978.106,E2 -11978.106} C_VEL
LIN {X 0,Y 534.575,Z 598.744,A -85,B 0,C 180,E1 -11979.428,E2 -11979.428} C_VEL
LIN {X 0,Y 535.009,Z 590.184,A -85,B 0,C 180,E1 -11980.563,E2 -11980.563} C_VEL
LIN {X 0,Y 535.595,Z 579.837,A -85,B 0,C 180,E1 -11981.697,E2 -11981.697} C_VEL
LIN {X 0,Y 536.174,Z 569.418,A -85,B 0,C 180,E1 -11982.641,E2 -11982.641} C_VEL
LIN {X 0,Y 536.951,Z 556.704,A -85,B 0,C 180,E1 -11983.582,E2 -11983.582} C_VEL
LIN {X 0,Y 537.615,Z 544.151,A -85,B 0,C 180,E1 -11984.334,E2 -11984.334} C_VEL
LIN {X 0,Y 538.388,Z 530.205,A -85,B 0,C 180,E1 -11984.987,E2 -11984.987} C_VEL
LIN {X 0,Y 538.909,Z 517.731,A -85,B 0,C 180,E1 -11985.43,E2 -11985.43} C_VEL
LIN {X 0,Y 539.37,Z 502.854,A -85,B 0,C 180,E1 -11985.803,E2 -11985.803} C_VEL
LIN {X 0,Y 541.598,Z 393.428,A -85,B 0,C 180,E1 -11987.602,E2 -11987.602} C_VEL
LIN {X 0,Y 538.923,Z 369.628,A -85,B 0,C 180,E1 -11988.154,E2 -11988.154} C_VEL
LIN {X 0,Y 536.448,Z 354.005,A -85,B 0,C 180,E1 -11988.582,E2 -11988.582} C_VEL
LIN {X 0,Y 536.28,Z 351.918,A -85,B 0,C 180,E1 -11988.679,E2 -11988.679} C_VEL
LIN {X 0,Y 537.47,Z 328.869,A -85,B 0,C 180,E1 -11991.805,E2 -11991.805} C_VEL
LIN {X 0,Y 538.597,Z 308.513,A -85,B 0,C 180,E1 -11994.594,E2 -11994.594} C_VEL
LIN {X 0,Y 535.473,Z 292.086,A -85,B 0,C 180,E1 -11997.036,E2 -11997.036} C_VEL
LIN {X 0,Y 535.151,Z 290.384,A -85,B 0,C 180,E1 -11997.319,E2 -11997.319} C_VEL
LIN {X 0,Y 535.083,Z 290.388,A -85,B 0,C 180,E1 -12000.235,E2 -12000.235} C_VEL
LIN {X 0,Y 535.036,Z 290.393,A -85,B 0,C 180,E1 -12003.085,E2 -12003.085} C_VEL
LIN {X 0,Y 535.077,Z 290.394,A -85,B 0,C 180,E1 -12005.746,E2 -12005.746} C_VEL
LIN {X 0,Y 535.037,Z 290.396,A -85,B 0,C 180,E1 -12008.933,E2 -12008.933} C_VEL
LIN {X 0,Y 535.053,Z 290.392,A -85,B 0,C 180,E1 -12011.887,E2 -12011.887} C_VEL
LIN {X 0,Y 535.101,Z 290.389,A -85,B 0,C 180,E1 -12015.02,E2 -12015.02} C_VEL
LIN {X 0,Y 535.054,Z 290.391,A -85,B 0,C 180,E1 -12018.114,E2 -12018.114} C_VEL
LIN {X 0,Y 535.039,Z 290.398,A -85,B 0,C 180,E1 -12021.068,E2 -12021.068} C_VEL
LIN {X 0,Y 535.1,Z 290.387,A -85,B 0,C 180,E1 -12023.91,E2 -12023.91} C_VEL
LIN {X 0,Y 535.073,Z 290.392,A -85,B 0,C 180,E1 -12026.91,E2 -12026.91} C_VEL
LIN {X 0,Y 535.089,Z 290.389,A -85,B 0,C 180,E1 -12029.766,E2 -12029.766} C_VEL
LIN {X 0,Y 535.108,Z 290.389,A -85,B 0,C 180,E1 -12032.733,E2 -12032.733} C_VEL
LIN {X 0,Y 535.103,Z 290.394,A -85,B 0,C 180,E1 -12036.059,E2 -12036.059} C_VEL
LIN {X 0,Y 535.141,Z 290.389,A -85,B 0,C 180,E1 -12039.304,E2 -12039.304} C_VEL
LIN {X 0,Y 535.1,Z 290.394,A -85,B 0,C 180,E1 -12041.69,E2 -12041.69} C_VEL
LIN {X 0,Y 535.125,Z 290.388,A -85,B 0,C 180,E1 -12044.045,E2 -12044.045} C_VEL
LIN {X 0,Y 535.214,Z 290.467,A -85,B 0,C 180,E1 -12046.109,E2 -12046.109} C_VEL
LIN {X 0,Y 538.718,Z 305.531,A -85,B 0,C 180,E1 -12048.373,E2 -12048.373} C_VEL
LIN {X 0,Y 539.449,Z 310.906,A -85,B 0,C 180,E1 -12049.148,E2 -12049.148} C_VEL
LIN {X 0,Y 538.787,Z 330.621,A -85,B 0,C 180,E1 -12051.778,E2 -12051.778} C_VEL
LIN {X 0,Y 538.172,Z 343.956,A -85,B 0,C 180,E1 -12053.555,E2 -12053.555} C_VEL
LIN {X 0,Y 541.99,Z 362.933,A -85,B 0,C 180,E1 -12054.077,E2 -12054.077} C_VEL
LIN {X 0,Y 542.443,Z 367.867,A -85,B 0,C 180,E1 -12054.187,E2 -12054.187} C_VEL
LIN {X 0,Y 540.051,Z 483.643,A -85,B 0,C 180,E1 -12056.096,E2 -12056.096} C_VEL
LIN {X 0,Y 539.587,Z 497.502,A -85,B 0,C 180,E1 -12056.465,E2 -12056.465} C_VEL
LIN {X 0,Y 538.91,Z 512.109,A -85,B 0,C 180,E1 -12057.02,E2 -12057.02} C_VEL
LIN {X 0,Y 538.272,Z 525.083,A -85,B 0,C 180,E1 -12057.669,E2 -12057.669} C_VEL
LIN {X 0,Y 537.457,Z 538.362,A -85,B 0,C 180,E1 -12058.506,E2 -12058.506} C_VEL
LIN {X 0,Y 536.787,Z 550.242,A -85,B 0,C 180,E1 -12059.439,E2 -12059.439} C_VEL
LIN {X 0,Y 536.029,Z 561.861,A -85,B 0,C 180,E1 -12060.562,E2 -12060.562} C_VEL
LIN {X 0,Y 535.284,Z 571.48,A -85,B 0,C 180,E1 -12061.687,E2 -12061.687} C_VEL
LIN {X 0,Y 534.829,Z 579.447,A -85,B 0,C 180,E1 -12062.815,E2 -12062.815} C_VEL
LIN {X 0,Y 534.367,Z 585.126,A -85,B 0,C 180,E1 -12063.758,E2 -12063.758} C_VEL
LIN {X 0,Y 534.245,Z 590.522,A -85,B 0,C 180,E1 -12064.833,E2 -12064.833} C_VEL
LIN {X 0,Y 534.01,Z 595.435,A -85,B 0,C 180,E1 -12066.023,E2 -12066.023} C_VEL
LIN {X 0,Y 533.746,Z 600.245,A -85,B 0,C 180,E1 -12067.541,E2 -12067.541} C_VEL
LIN {X 0,Y 533.616,Z 603.478,A -85,B 0,C 180,E1 -12069.063,E2 -12069.063} C_VEL
LIN {X 0,Y 533.569,Z 605.242,A -85,B 0,C 180,E1 -12070.59,E2 -12070.59} C_VEL
LIN {X 0,Y 533.454,Z 605.579,A -85,B 0,C 180,E1 -12072.127,E2 -12072.127} C_VEL
LIN {X 0,Y 533.572,Z 604.4,A -85,B 0,C 180,E1 -12073.725,E2 -12073.725} C_VEL
LIN {X 0,Y 533.55,Z 601.857,A -85,B 0,C 180,E1 -12075.222,E2 -12075.222} C_VEL
LIN {X 0,Y 533.73,Z 598.024,A -85,B 0,C 180,E1 -12076.657,E2 -12076.657} C_VEL
LIN {X 0,Y 533.845,Z 593.305,A -85,B 0,C 180,E1 -12077.959,E2 -12077.959} C_VEL
LIN {X 0,Y 534.097,Z 587.48,A -85,B 0,C 180,E1 -12079.22,E2 -12079.22} C_VEL
LIN {X 0,Y 534.358,Z 579.955,A -85,B 0,C 180,E1 -12080.527,E2 -12080.527} C_VEL
LIN {X 0,Y 534.77,Z 571.723,A -85,B 0,C 180,E1 -12081.696,E2 -12081.696} C_VEL
LIN {X 0,Y 535.258,Z 561.322,A -85,B 0,C 180,E1 -12082.912,E2 -12082.912} C_VEL
LIN {X 0,Y 535.787,Z 550.979,A -85,B 0,C 180,E1 -12083.908,E2 -12083.908} C_VEL
LIN {X 0,Y 536.318,Z 539.737,A -85,B 0,C 180,E1 -12084.807,E2 -12084.807} C_VEL
LIN {X 0,Y 536.835,Z 527.421,A -85,B 0,C 180,E1 -12085.615,E2 -12085.615} C_VEL
LIN {X 0,Y 537.385,Z 514.121,A -85,B 0,C 180,E1 -12086.306,E2 -12086.306} C_VEL
LIN {X 0,Y 537.868,Z 500.418,A -85,B 0,C 180,E1 -12086.854,E2 -12086.854} C_VEL
LIN {X 0,Y 538.321,Z 485.816,A -85,B 0,C 180,E1 -12087.275,E2 -12087.275} C_VEL
LIN {X 0,Y 538.597,Z 470.964,A -85,B 0,C 180,E1 -12087.548,E2 -12087.548} C_VEL
LIN {X 0,Y 540.005,Z 364.534,A -85,B 0,C 180,E1 -12089.174,E2 -12089.174} C_VEL
LIN {X 0,Y 536.762,Z 342.694,A -85,B 0,C 180,E1 -12089.626,E2 -12089.626} C_VEL
LIN {X 0,Y 537.473,Z 321.268,A -85,B 0,C 180,E1 -12092.519,E2 -12092.519} C_VEL
LIN {X 0,Y 538.019,Z 306.652,A -85,B 0,C 180,E1 -12094.494,E2 -12094.494} C_VEL
LIN {X 0,Y 536.945,Z 299.641,A -85,B 0,C 180,E1 -12095.486,E2 -12095.486} C_VEL
LIN {X 0,Y 535.159,Z 290.383,A -85,B 0,C 180,E1 -12096.826,E2 -12096.826} C_VEL
LIN {X 0,Y 535.079,Z 290.392,A -85,B 0,C 180,E1 -12099.899,E2 -12099.899} C_VEL
LIN {X 0,Y 535.093,Z 290.388,A -85,B 0,C 180,E1 -12102.897,E2 -12102.897} C_VEL
LIN {X 0,Y 535.104,Z 290.391,A -85,B 0,C 180,E1 -12106.07,E2 -12106.07} C_VEL
LIN {X 0,Y 535.063,Z 290.391,A -85,B 0,C 180,E1 -12109.4,E2 -12109.4} C_VEL
LIN {X 0,Y 535.031,Z 290.399,A -85,B 0,C 180,E1 -12112.024,E2 -12112.024} C_VEL
LIN {X 0,Y 535.064,Z 290.393,A -85,B 0,C 180,E1 -12114.829,E2 -12114.829} C_VEL
LIN {X 0,Y 535.055,Z 290.394,A -85,B 0,C 180,E1 -12117.537,E2 -12117.537} C_VEL
LIN {X 0,Y 535.088,Z 290.39,A -85,B 0,C 180,E1 -12120.168,E2 -12120.168} C_VEL
LIN {X 0,Y 535.092,Z 290.388,A -85,B 0,C 180,E1 -12122.89,E2 -12122.89} C_VEL
LIN {X 0,Y 535.1,Z 290.389,A -85,B 0,C 180,E1 -12126.058,E2 -12126.058} C_VEL
LIN {X 0,Y 535.139,Z 290.382,A -85,B 0,C 180,E1 -12129.303,E2 -12129.303} C_VEL
LIN {X 0,Y 535.12,Z 290.385,A -85,B 0,C 180,E1 -12132.477,E2 -12132.477} C_VEL
LIN {X 0,Y 535.167,Z 290.377,A -85,B 0,C 180,E1 -12134.823,E2 -12134.823} C_VEL
LIN {X 0,Y 535.168,Z 290.377,A -85,B 0,C 180,E1 -12137.142,E2 -12137.142} C_VEL
LIN {X 0,Y 535.151,Z 290.383,A -85,B 0,C 180,E1 -12138.047,E2 -12138.047} C_VEL
LIN {X 0,Y 534.493,Z 290.461,A -85,B 0,C 180,E1 -12138.675,E2 -12138.675} C_VEL
LIN {X 0,Y 531.636,Z 290.821,A -85,B 0,C 180,E1 -12139.696,E2 -12139.696} C_VEL
LIN {X 0,Y 529.232,Z 291.121,A -85,B 0,C 180,E1 -12140.517,E2 -12140.517} C_VEL
LIN {X 0,Y 528.225,Z 291.245,A -85,B 0,C 180,E1 -12141.152,E2 -12141.152} C_VEL
LIN {X 0,Y 528.157,Z 291.254,A -85,B 0,C 180,E1 -12141.366,E2 -12141.366} C_VEL
LIN {X 0,Y 528.243,Z 291.338,A -85,B 0,C 180,E1 -12142.235,E2 -12142.235} C_VEL
LIN {X 0,Y 529.6,Z 299.973,A -85,B 0,C 180,E1 -12143.925,E2 -12143.925} C_VEL
LIN {X 0,Y 529.679,Z 301.99,A -85,B 0,C 180,E1 -12144.306,E2 -12144.306} C_VEL
LIN {X 0,Y 533.56,Z 321.809,A -85,B 0,C 180,E1 -12144.702,E2 -12144.702} C_VEL
LIN {X 0,Y 532.262,Z 437.574,A -85,B 0,C 180,E1 -12146.273,E2 -12146.273} C_VEL
LIN {X 0,Y 531.951,Z 452.028,A -85,B 0,C 180,E1 -12146.625,E2 -12146.625} C_VEL
LIN {X 0,Y 531.527,Z 465.858,A -85,B 0,C 180,E1 -12147.118,E2 -12147.118} C_VEL
LIN {X 0,Y 531.064,Z 478.714,A -85,B 0,C 180,E1 -12147.731,E2 -12147.731} C_VEL
LIN {X 0,Y 530.565,Z 491.175,A -85,B 0,C 180,E1 -12148.485,E2 -12148.485} C_VEL
LIN {X 0,Y 529.779,Z 502.63,A -85,B 0,C 180,E1 -12149.335,E2 -12149.335} C_VEL
LIN {X 0,Y 529.283,Z 514.027,A -85,B 0,C 180,E1 -12150.377,E2 -12150.377} C_VEL
LIN {X 0,Y 528.555,Z 524.3,A -85,B 0,C 180,E1 -12151.517,E2 -12151.517} C_VEL
LIN {X 0,Y 528.099,Z 532.758,A -85,B 0,C 180,E1 -12152.659,E2 -12152.659} C_VEL
LIN {X 0,Y 527.539,Z 540.883,A -85,B 0,C 180,E1 -12153.995,E2 -12153.995} C_VEL
LIN {X 0,Y 527.355,Z 547.402,A -85,B 0,C 180,E1 -12155.333,E2 -12155.333} C_VEL
LIN {X 0,Y 527.033,Z 553.224,A -85,B 0,C 180,E1 -12156.868,E2 -12156.868} C_VEL
LIN {X 0,Y 526.771,Z 557.493,A -85,B 0,C 180,E1 -12158.409,E2 -12158.409} C_VEL
LIN {X 0,Y 526.75,Z 560.315,A -85,B 0,C 180,E1 -12159.953,E2 -12159.953} C_VEL
LIN {X 0,Y 526.662,Z 561.783,A -85,B 0,C 180,E1 -12161.505,E2 -12161.505} C_VEL
LIN {X 0,Y 526.732,Z 561.896,A -85,B 0,C 180,E1 -12163.063,E2 -12163.063} C_VEL
LIN {X 0,Y 526.846,Z 560.636,A -85,B 0,C 180,E1 -12164.63,E2 -12164.63} C_VEL
LIN {X 0,Y 526.998,Z 557.946,A -85,B 0,C 180,E1 -12166.205,E2 -12166.205} C_VEL
LIN {X 0,Y 527.298,Z 553.746,A -85,B 0,C 180,E1 -12167.787,E2 -12167.787} C_VEL
LIN {X 0,Y 527.701,Z 549.538,A -85,B 0,C 180,E1 -12168.975,E2 -12168.975} C_VEL
LIN {X 0,Y 528.16,Z 543.279,A -85,B 0,C 180,E1 -12170.37,E2 -12170.37} C_VEL
LIN {X 0,Y 528.809,Z 535.382,A -85,B 0,C 180,E1 -12171.767,E2 -12171.767} C_VEL
LIN {X 0,Y 529.525,Z 527.056,A -85,B 0,C 180,E1 -12172.966,E2 -12172.966} C_VEL
LIN {X 0,Y 530.37,Z 516.922,A -85,B 0,C 180,E1 -12174.165,E2 -12174.165} C_VEL
LIN {X 0,Y 531.143,Z 506.651,A -85,B 0,C 180,E1 -12175.167,E2 -12175.167} C_VEL
LIN {X 0,Y 532.041,Z 494.373,A -85,B 0,C 180,E1 -12176.148,E2 -12176.148} C_VEL
LIN {X 0,Y 532.694,Z 483.245,A -85,B 0,C 180,E1 -12176.87,E2 -12176.87} C_VEL
LIN {X 0,Y 533.397,Z 470.768,A -85,B 0,C 180,E1 -12177.518,E2 -12177.518} C_VEL
LIN {X 0,Y 533.886,Z 458.325,A -85,B 0,C 180,E1 -12178.022,E2 -12178.022} C_VEL
LIN {X 0,Y 534.26,Z 443.9,A -85,B 0,C 180,E1 -12178.445,E2 -12178.445} C_VEL
LIN {X 0,Y 534.452,Z 428.484,A -85,B 0,C 180,E1 -12178.721,E2 -12178.721} C_VEL
LIN {X 0,Y 535.752,Z 322.087,A -85,B 0,C 180,E1 -12180.172,E2 -12180.172} C_VEL
LIN {X 0,Y 532.041,Z 307.472,A -85,B 0,C 180,E1 -12180.537,E2 -12180.537} C_VEL
LIN {X 0,Y 530.274,Z 302.646,A -85,B 0,C 180,E1 -12180.697,E2 -12180.697} C_VEL
LIN {X 0,Y 528.006,Z 291.272,A -85,B 0,C 180,E1 -12183.104,E2 -12183.104} C_VEL
LIN {X 0,Y 528.011,Z 291.275,A -85,B 0,C 180,E1 -12185.981,E2 -12185.981} C_VEL
LIN {X 0,Y 527.982,Z 291.271,A -85,B 0,C 180,E1 -12188.571,E2 -12188.571} C_VEL
LIN {X 0,Y 528.002,Z 291.267,A -85,B 0,C 180,E1 -12191.548,E2 -12191.548} C_VEL
LIN {X 0,Y 528.018,Z 291.258,A -85,B 0,C 180,E1 -12194.671,E2 -12194.671} C_VEL
LIN {X 0,Y 528.03,Z 291.269,A -85,B 0,C 180,E1 -12197.427,E2 -12197.427} C_VEL
LIN {X 0,Y 527.999,Z 291.271,A -85,B 0,C 180,E1 -12200.449,E2 -12200.449} C_VEL
LIN {X 0,Y 528.053,Z 291.258,A -85,B 0,C 180,E1 -12203.351,E2 -12203.351} C_VEL
LIN {X 0,Y 527.994,Z 291.273,A -85,B 0,C 180,E1 -12206.139,E2 -12206.139} C_VEL
LIN {X 0,Y 528.012,Z 291.264,A -85,B 0,C 180,E1 -12208.845,E2 -12208.845} C_VEL
LIN {X 0,Y 528.024,Z 291.272,A -85,B 0,C 180,E1 -12211.474,E2 -12211.474} C_VEL
LIN {X 0,Y 528.013,Z 291.268,A -85,B 0,C 180,E1 -12214.425,E2 -12214.425} C_VEL
LIN {X 0,Y 528.021,Z 291.264,A -85,B 0,C 180,E1 -12217.375,E2 -12217.375} C_VEL
LIN {X 0,Y 528.068,Z 291.256,A -85,B 0,C 180,E1 -12220.342,E2 -12220.342} C_VEL
LIN {X 0,Y 528.066,Z 291.262,A -85,B 0,C 180,E1 -12223.033,E2 -12223.033} C_VEL
LIN {X 0,Y 528.125,Z 291.247,A -85,B 0,C 180,E1 -12226.188,E2 -12226.188} C_VEL
LIN {X 0,Y 528.155,Z 291.254,A -85,B 0,C 180,E1 -12229.3,E2 -12229.3} C_VEL
LIN {X 0,Y 528.177,Z 291.244,A -85,B 0,C 180,E1 -12232.379,E2 -12232.379} C_VEL
LIN {X 0,Y 528.214,Z 291.244,A -85,B 0,C 180,E1 -12234.674,E2 -12234.674} C_VEL
LIN {X 0,Y 528.236,Z 291.229,A -85,B 0,C 180,E1 -12236.199,E2 -12236.199} C_VEL
LIN {X 0,Y 528.358,Z 291.23,A -85,B 0,C 180,E1 -12239.24,E2 -12239.24} C_VEL
LIN {X 0,Y 528.215,Z 291.234,A -85,B 0,C 180,E1 -12241.52,E2 -12241.52} C_VEL
LIN {X 0,Y 528.264,Z 291.238,A -85,B 0,C 180,E1 -12244.563,E2 -12244.563} C_VEL
LIN {X 0,Y 528.197,Z 291.241,A -85,B 0,C 180,E1 -12246.855,E2 -12246.855} C_VEL
LIN {X 0,Y 528.151,Z 291.248,A -85,B 0,C 180,E1 -12249.928,E2 -12249.928} C_VEL
LIN {X 0,Y 528.122,Z 291.247,A -85,B 0,C 180,E1 -12252.252,E2 -12252.252} C_VEL
LIN {X 0,Y 528.144,Z 291.252,A -85,B 0,C 180,E1 -12254.595,E2 -12254.595} C_VEL
LIN {X 0,Y 528.068,Z 291.25,A -85,B 0,C 180,E1 -12257.763,E2 -12257.763} C_VEL
LIN {X 0,Y 528.068,Z 291.261,A -85,B 0,C 180,E1 -12260.174,E2 -12260.174} C_VEL
LIN {X 0,Y 528.022,Z 291.264,A -85,B 0,C 180,E1 -12262.625,E2 -12262.625} C_VEL
LIN {X 0,Y 528.013,Z 291.264,A -85,B 0,C 180,E1 -12265.575,E2 -12265.575} C_VEL
LIN {X 0,Y 528.025,Z 291.273,A -85,B 0,C 180,E1 -12268.526,E2 -12268.526} C_VEL
LIN {X 0,Y 528.05,Z 291.263,A -85,B 0,C 180,E1 -12271.153,E2 -12271.153} C_VEL
LIN {X 0,Y 528.036,Z 291.264,A -85,B 0,C 180,E1 -12273.858,E2 -12273.858} C_VEL
LIN {X 0,Y 528.101,Z 291.245,A -85,B 0,C 180,E1 -12276.645,E2 -12276.645} C_VEL
LIN {X 0,Y 528.056,Z 291.263,A -85,B 0,C 180,E1 -12279.709,E2 -12279.709} C_VEL
LIN {X 0,Y 528.041,Z 291.266,A -85,B 0,C 180,E1 -12282.572,E2 -12282.572} C_VEL
LIN {X 0,Y 528.029,Z 291.263,A -85,B 0,C 180,E1 -12285.331,E2 -12285.331} C_VEL
LIN {X 0,Y 528.075,Z 291.264,A -85,B 0,C 180,E1 -12288.459,E2 -12288.459} C_VEL
LIN {X 0,Y 528.056,Z 291.264,A -85,B 0,C 180,E1 -12291.5,E2 -12291.5} C_VEL
LIN {X 0,Y 528.078,Z 291.264,A -85,B 0,C 180,E1 -12294.298,E2 -12294.298} C_VEL
LIN {X 0,Y 528.026,Z 291.273,A -85,B 0,C 180,E1 -12297.055,E2 -12297.055} C_VEL
LIN {X 0,Y 528.044,Z 291.275,A -85,B 0,C 180,E1 -12299.733,E2 -12299.733} C_VEL
LIN {X 0,Y 528.066,Z 291.298,A -85,B 0,C 180,E1 -12301.245,E2 -12301.245} C_VEL
LIN {X 0,Y 531.379,Z 305.982,A -85,B 0,C 180,E1 -12303.683,E2 -12303.683} C_VEL
LIN {X 0,Y 532.894,Z 313.887,A -85,B 0,C 180,E1 -12304.942,E2 -12304.942} C_VEL
LIN {X 0,Y 531.601,Z 331.905,A -85,B 0,C 180,E1 -12307.538,E2 -12307.538} C_VEL
LIN {X 0,Y 530.115,Z 354.342,A -85,B 0,C 180,E1 -12310.714,E2 -12310.714} C_VEL
LIN {X 0,Y 529.845,Z 358.979,A -85,B 0,C 180,E1 -12311.347,E2 -12311.347} C_VEL
LIN {X 0,Y 534.054,Z 385.176,A -85,B 0,C 180,E1 -12311.892,E2 -12311.892} C_VEL
LIN {X 0,Y 535.123,Z 393.997,A -85,B 0,C 180,E1 -12312.059,E2 -12312.059} C_VEL
LIN {X 0,Y 533.802,Z 497.645,A -85,B 0,C 180,E1 -12313.49,E2 -12313.49} C_VEL
LIN {X 0,Y 533.201,Z 512.307,A -85,B 0,C 180,E1 -12313.848,E2 -12313.848} C_VEL
LIN {X 0,Y 532.417,Z 526.476,A -85,B 0,C 180,E1 -12314.356,E2 -12314.356} C_VEL
LIN {X 0,Y 531.658,Z 538.375,A -85,B 0,C 180,E1 -12314.92,E2 -12314.92} C_VEL
LIN {X 0,Y 530.812,Z 550.999,A -85,B 0,C 180,E1 -12315.677,E2 -12315.677} C_VEL
LIN {X 0,Y 529.856,Z 562.525,A -85,B 0,C 180,E1 -12316.529,E2 -12316.529} C_VEL
LIN {X 0,Y 528.956,Z 574.109,A -85,B 0,C 180,E1 -12317.576,E2 -12317.576} C_VEL
LIN {X 0,Y 528.313,Z 584.5,A -85,B 0,C 180,E1 -12318.724,E2 -12318.724} C_VEL
LIN {X 0,Y 527.632,Z 593.111,A -85,B 0,C 180,E1 -12319.871,E2 -12319.871} C_VEL
LIN {X 0,Y 527.141,Z 601.397,A -85,B 0,C 180,E1 -12321.212,E2 -12321.212} C_VEL
LIN {X 0,Y 526.763,Z 608.927,A -85,B 0,C 180,E1 -12322.745,E2 -12322.745} C_VEL
LIN {X 0,Y 526.65,Z 614.242,A -85,B 0,C 180,E1 -12323.894,E2 -12323.894} C_VEL
LIN {X 0,Y 526.591,Z 618.599,A -85,B 0,C 180,E1 -12325.042,E2 -12325.042} C_VEL
LIN {X 0,Y 526.539,Z 622.029,A -85,B 0,C 180,E1 -12326.188,E2 -12326.188} C_VEL
LIN {X 0,Y 526.57,Z 625.19,A -85,B 0,C 180,E1 -12327.715,E2 -12327.715} C_VEL
LIN {X 0,Y 526.565,Z 626.887,A -85,B 0,C 180,E1 -12329.24,E2 -12329.24} C_VEL
LIN {X 0,Y 526.558,Z 627.153,A -85,B 0,C 180,E1 -12330.764,E2 -12330.764} C_VEL
LIN {X 0,Y 526.57,Z 625.995,A -85,B 0,C 180,E1 -12332.289,E2 -12332.289} C_VEL
LIN {X 0,Y 526.549,Z 623.233,A -85,B 0,C 180,E1 -12333.893,E2 -12333.893} C_VEL
LIN {X 0,Y 526.642,Z 619.269,A -85,B 0,C 180,E1 -12335.344,E2 -12335.344} C_VEL
LIN {X 0,Y 526.791,Z 613.497,A -85,B 0,C 180,E1 -12336.875,E2 -12336.875} C_VEL
LIN {X 0,Y 527.034,Z 606.971,A -85,B 0,C 180,E1 -12338.216,E2 -12338.216} C_VEL
LIN {X 0,Y 527.547,Z 598.834,A -85,B 0,C 180,E1 -12339.555,E2 -12339.555} C_VEL
LIN {X 0,Y 528.039,Z 590.311,A -85,B 0,C 180,E1 -12340.704,E2 -12340.704} C_VEL
LIN {X 0,Y 528.65,Z 580.05,A -85,B 0,C 180,E1 -12341.853,E2 -12341.853} C_VEL
LIN {X 0,Y 529.315,Z 568.556,A -85,B 0,C 180,E1 -12342.905,E2 -12342.905} C_VEL
LIN {X 0,Y 530.157,Z 555.724,A -85,B 0,C 180,E1 -12343.857,E2 -12343.857} C_VEL
LIN {X 0,Y 530.93,Z 542.975,A -85,B 0,C 180,E1 -12344.616,E2 -12344.616} C_VEL
LIN {X 0,Y 531.662,Z 529.873,A -85,B 0,C 180,E1 -12345.23,E2 -12345.23} C_VEL
LIN {X 0,Y 532.131,Z 518.139,A -85,B 0,C 180,E1 -12345.656,E2 -12345.656} C_VEL
LIN {X 0,Y 532.651,Z 503.8,A -85,B 0,C 180,E1 -12346.032,E2 -12346.032} C_VEL
LIN {X 0,Y 534.968,Z 393.34,A -85,B 0,C 180,E1 -12347.897,E2 -12347.897} C_VEL
LIN {X 0,Y 532.453,Z 371.014,A -85,B 0,C 180,E1 -12348.43,E2 -12348.43} C_VEL
LIN {X 0,Y 529.809,Z 353.95,A -85,B 0,C 180,E1 -12348.906,E2 -12348.906} C_VEL
LIN {X 0,Y 529.367,Z 350.242,A -85,B 0,C 180,E1 -12349.07,E2 -12349.07} C_VEL
LIN {X 0,Y 530.641,Z 327.131,A -85,B 0,C 180,E1 -12352.249,E2 -12352.249} C_VEL
LIN {X 0,Y 531.636,Z 310.068,A -85,B 0,C 180,E1 -12354.62,E2 -12354.62} C_VEL
LIN {X 0,Y 529.253,Z 297.29,A -85,B 0,C 180,E1 -12356.537,E2 -12356.537} C_VEL
LIN {X 0,Y 528.122,Z 291.261,A -85,B 0,C 180,E1 -12357.47,E2 -12357.47} C_VEL
LIN {X 0,Y 528.049,Z 291.265,A -85,B 0,C 180,E1 -12360.434,E2 -12360.434} C_VEL
LIN {X 0,Y 528.003,Z 291.271,A -85,B 0,C 180,E1 -12363.306,E2 -12363.306} C_VEL
LIN {X 0,Y 528.022,Z 291.272,A -85,B 0,C 180,E1 -12365.983,E2 -12365.983} C_VEL
LIN {X 0,Y 527.998,Z 291.271,A -85,B 0,C 180,E1 -12368.574,E2 -12368.574} C_VEL
LIN {X 0,Y 528.015,Z 291.271,A -85,B 0,C 180,E1 -12370.875,E2 -12370.875} C_VEL
LIN {X 0,Y 528.029,Z 291.268,A -85,B 0,C 180,E1 -12373.615,E2 -12373.615} C_VEL
LIN {X 0,Y 528.047,Z 291.265,A -85,B 0,C 180,E1 -12376.388,E2 -12376.388} C_VEL
LIN {X 0,Y 528.016,Z 291.27,A -85,B 0,C 180,E1 -12379.457,E2 -12379.457} C_VEL
LIN {X 0,Y 528.054,Z 291.268,A -85,B 0,C 180,E1 -12382.74,E2 -12382.74} C_VEL
LIN {X 0,Y 528.027,Z 291.268,A -85,B 0,C 180,E1 -12385.333,E2 -12385.333} C_VEL
LIN {X 0,Y 528.014,Z 291.271,A -85,B 0,C 180,E1 -12388.105,E2 -12388.105} C_VEL
LIN {X 0,Y 528.057,Z 291.264,A -85,B 0,C 180,E1 -12391.102,E2 -12391.102} C_VEL
LIN {X 0,Y 528.052,Z 291.269,A -85,B 0,C 180,E1 -12394.04,E2 -12394.04} C_VEL
LIN {X 0,Y 528.054,Z 291.273,A -85,B 0,C 180,E1 -12396.551,E2 -12396.551} C_VEL
LIN {X 0,Y 528.085,Z 291.268,A -85,B 0,C 180,E1 -12399.015,E2 -12399.015} C_VEL
LIN {X 0,Y 528.057,Z 291.271,A -85,B 0,C 180,E1 -12401.437,E2 -12401.437} C_VEL
LIN {X 0,Y 528.07,Z 291.268,A -85,B 0,C 180,E1 -12403.826,E2 -12403.826} C_VEL
LIN {X 0,Y 528.183,Z 291.374,A -85,B 0,C 180,E1 -12405.77,E2 -12405.77} C_VEL
